// ---- __TESTs/MessagesTests/Complex/FB_ComplexDataTests.TcPOU
FUNCTION_BLOCK INTERNAL FINAL FB_ComplexDataTests EXTENDS FB_TestSuite
VAR
	fbVerify			: FB_TcUnitAdapter;
	fbVerifyBuffer 		: FB_TcUnitAdapter;
	fbWriterSUT			: FB_ComplexData;
	fbParserSUT			: FB_ComplexData;
	stActual			: ST_ComplexData;
	aBuffer				: ARRAY[0..255] OF BYTE;
	eTestState			: (DATA, BUFFER);
END_VAR
VAR CONSTANT
	cExpected			: ST_ComplexData := (label:= 'test-label 🐞!', value_dint:= -1, value_int:= -2, value_word:= 2,
											raw_bytes:= [44,33,22], raw_bytes_count:= 3,
											readings:= [(value:= 12345.67892, precision:= 2.3, timestamp:= 12345678), (value:= 999.888, precision:= 0.111, timestamp:= 777666555)], readings_count:= 2,
											data_type:= E_DataType.DATA_TYPE_TEMPERATURE);
END_VAR

VerifyData();
VerifyBuffer();

METHOD PRIVATE VerifyBuffer
VAR
	hr : HRESULT;
END_VAR
TEST(__POUNAME());

IF eTestState <> BUFFER THEN
	RETURN;
END_IF

hr := fbVerifyBuffer.Verify(anyArg:= aBuffer);

IF NOT PENDING(hr) THEN	
	TEST_FINISHED_NAMED(__POUNAME());
END_IF
END_METHOD

METHOD PRIVATE VerifyData
VAR_INST
	hr, hrWriter, hrParser : HRESULT;
	bOnce : BOOL := TRUE;
END_VAR
TEST(__POUNAME());
IF eTestState <> DATA THEN
	RETURN;
END_IF

// ARRANGE
fbWriterSUT.ComplexData := cExpected;

// ACT
IF bOnce THEN
	bOnce := FALSE;
	hrWriter := fbWriterSUT.Writer.WriteTo(aBuffer);
	hrParser := fbParserSUT.Parser.ParseFrom(aBuffer);
	stActual := fbParserSUT.ComplexData;
END_IF;

// ASSERT
hr := fbVerify.Verify(anyArg:= stActual);

IF NOT PENDING(hr) THEN
	AssertEquals_DINT(Expected:= 0, Actual:= hrWriter, Message:= 'Writer failed');
	AssertEquals_DINT(Expected:= 0, Actual:= hrParser, Message:= 'Parser failed');
	TEST_FINISHED_NAMED(__POUNAME());
	eTestState := BUFFER;
END_IF
END_METHOD

END_FUNCTION_BLOCK

// ---- __TESTs/MessagesTests/Complex/_gen/FB_ComplexData.TcPOU
(*******************************************************************************
                          protoc-gen-twincat V0.0.0.0                           
                  https://github.com/TcHaxx/protoc-gen-twincat                  
*******************************************************************************)
{attribute 'no_explicit_call' := 'do not call this POU directly'}
{attribute 'no-analysis'}
// Another message demonstrating all field options
FUNCTION_BLOCK INTERNAL FINAL FB_ComplexData IMPLEMENTS I_Message
VAR
    _fbMessageParser : FB_MessageParser(ipMessage:= THIS^);
    _fbMessageWriter : FB_MessageWriter(ipMessage:= THIS^);
    _stComplexData : ST_ComplexData;
    // repeated uint32 array_data = 5;
    _fbFieldCodecId5 : FB_FieldCodecUint32(nTag:= 16#2A);
    _fbRepeatedId5 : FB_RepeatedField(anyArray:= F_ToAnyType(_stComplexData.array_data), anyFirstElem:= F_ToAnyType(_stComplexData.array_data[0]), ipFieldCodec:= _fbFieldCodecId5);
    // repeated SensorReading readings = 10;
    _fbFieldCodecId10 : FB_FieldCodecMessage(nTag:= 16#52, ipMessage:= _fbreadings);
    _fbRepeatedId10 : FB_RepeatedField(anyArray:= F_ToAnyType(_stComplexData.readings), anyFirstElem:= F_ToAnyType(_stComplexData.readings[0]), ipFieldCodec:= _fbFieldCodecId10);
    _fbreadings : FB_SensorReading;
    END_VAR

{attribute 'no-analysis'}
(* Calculates the size of this message in Protocol Buffer wire format, in bytes. *)
METHOD CalculateSize : UDINT
VAR
    nSize : UDINT;
    nRepeatedFieldSize : UDINT;
END_VAR
// string label = 1;
nSize := nSize + 1 + F_ComputeStringSize(anyString:= _stComplexData.label);
// int32 value_dint = 2;
nSize := nSize + 1 + F_ComputeInt32Size(anyDint:= _stComplexData.value_dint);
// int32 value_int = 3;
nSize := nSize + 1 + F_ComputeInt32Size(anyDint:= _stComplexData.value_int);
// uint32 value_word = 4;
nSize := nSize + 1 + F_ComputeUint32Size(anyUdint:= _stComplexData.value_word);
// repeated uint32 array_data = 5;
_fbRepeatedId5.nCount := _stComplexData.array_data_count;
_fbRepeatedId5.CalculateSize(nSize => nRepeatedFieldSize);
nSize := nSize + nRepeatedFieldSize;
// Status state = 6;
nSize := nSize + 1 + F_ComputeEnumSize(anyEnum:= _stComplexData.state);
// bytes raw_bytes = 7;
nSize := nSize + 1 + F_ComputeBytesSize(aBytes:= _stComplexData.raw_bytes, nCount:= _stComplexData.raw_bytes_count);
// double measurement = 8;
nSize := nSize + 1 + F_ComputeDoubleSize(fValue:= _stComplexData.measurement);
// float calibration_factor = 9;
nSize := nSize + 1 + F_ComputeFloatSize(fValue:= _stComplexData.calibration_factor);
// repeated SensorReading readings = 10;
_fbRepeatedId10.nCount := _stComplexData.readings_count;
_fbRepeatedId10.CalculateSize(nSize => nRepeatedFieldSize);
nSize := nSize + nRepeatedFieldSize;
// DataType data_type = 11;
nSize := nSize + 1 + F_ComputeEnumSize(anyEnum:= _stComplexData.data_type);
CalculateSize := nSize;
END_METHOD

PROPERTY PUBLIC ComplexData : ST_ComplexData
GET
ComplexData := _stComplexData;
END_GET
SET
_stComplexData := ComplexData;
// repeated SensorReading readings = 10;
_stComplexData.readings := ComplexData.readings;
END_SET
END_PROPERTY

(* Merges the data from the specified coded input stream with the current message.*)
{attribute 'no-analysis'}
METHOD MergeFrom : HRESULT
VAR_IN_OUT
    fbParseCtx : FB_ParseContext;
END_VAR
VAR
    nTag : UDINT;
END_VAR
_fbRepeatedId10.Initialize();
_fbRepeatedId5.Initialize();
REPEAT
MergeFrom := fbParseCtx.ReadTag(nTag=> nTag);
IF SUCCEEDED(MergeFrom) AND nTag = 0 THEN
    EXIT;
END_IF;

IF FAILED(MergeFrom) THEN
    RETURN;
END_IF

CASE nTag OF
    16#0A:    // string label = 1;
        MergeFrom := fbParseCtx.ReadString(anyStringOut:= _stComplexData.label); 
    16#10:    // int32 value_dint = 2;
        MergeFrom := fbParseCtx.ReadInt32(anyDint:= _stComplexData.value_dint); 
    16#18:    // int32 value_int = 3;
        MergeFrom := fbParseCtx.ReadInt32(anyDint:= _stComplexData.value_int); 
    16#20:    // uint32 value_word = 4;
        MergeFrom := fbParseCtx.ReadUint32(anyUdint:= _stComplexData.value_word); 
    16#2A:    // repeated uint32 array_data = 5;
        MergeFrom := _fbRepeatedId5.AddEntriesFrom(fbParseCtx:= fbParseCtx, ipFieldCodec:= _fbFieldCodecId5,nCount=> _stComplexData.array_data_count);
    16#30:    // Status state = 6;
        MergeFrom := fbParseCtx.ReadEnum(anyEnum:= _stComplexData.state); 
    16#3A:    // bytes raw_bytes = 7;
        MergeFrom := fbParseCtx.ReadBytes(aBytes:= _stComplexData.raw_bytes, nCount=> _stComplexData.raw_bytes_count); 
    16#41:    // double measurement = 8;
        MergeFrom := fbParseCtx.ReadDouble(fValue=> _stComplexData.measurement); 
    16#4D:    // float calibration_factor = 9;
        MergeFrom := fbParseCtx.ReadFloat(fValue=> _stComplexData.calibration_factor); 
    16#52:    // repeated SensorReading readings = 10;
        MergeFrom := _fbRepeatedId10.AddEntriesFrom(fbParseCtx:= fbParseCtx, ipFieldCodec:= _fbFieldCodecId10,nCount=> _stComplexData.readings_count);
    16#58:    // DataType data_type = 11;
        MergeFrom := fbParseCtx.ReadEnum(anyEnum:= _stComplexData.data_type); 
ELSE
    MergeFrom := fbParseCtx.SkipLastField();
END_CASE

UNTIL (FAILED(MergeFrom) OR nTag = 0)
END_REPEAT
END_METHOD

PROPERTY PUBLIC MessageValue : T_Any
GET
MessageValue := F_ToAnyType(anyArg:= _stComplexData);
END_GET
END_PROPERTY

PROPERTY PUBLIC Parser : REFERENCE TO FB_MessageParser
GET
Parser REF= THIS^._fbMessageParser;
END_GET
END_PROPERTY

(* Writer for this message.*)
PROPERTY PUBLIC Writer : REFERENCE TO FB_MessageWriter
GET
Writer REF= THIS^._fbMessageWriter;
END_GET
END_PROPERTY

(* Writes the data to the given coded output stream.*)
{attribute 'no-analysis'}
METHOD WriteTo : HRESULT
VAR_IN_OUT
	(* Coded output stream to write the data to. *)
	fbWriteCtx	: FB_WriteContext;
END_VAR
// string label = 1;
WriteTo := fbWriteCtx.WriteTag(1, E_WireType.LengthDelimited);
IF FAILED(WriteTo) THEN
    RETURN;
END_IF
WriteTo := fbWriteCtx.WriteString(sStringToWrite:= _stComplexData.label);
IF FAILED(WriteTo) THEN
    RETURN;
END_IF
// int32 value_dint = 2;
WriteTo := fbWriteCtx.WriteTag(2, E_WireType.Varint);
IF FAILED(WriteTo) THEN
    RETURN;
END_IF
WriteTo := fbWriteCtx.WriteInt32(anyDint:= _stComplexData.value_dint);
IF FAILED(WriteTo) THEN
    RETURN;
END_IF
// int32 value_int = 3;
WriteTo := fbWriteCtx.WriteTag(3, E_WireType.Varint);
IF FAILED(WriteTo) THEN
    RETURN;
END_IF
WriteTo := fbWriteCtx.WriteInt32(anyDint:= _stComplexData.value_int);
IF FAILED(WriteTo) THEN
    RETURN;
END_IF
// uint32 value_word = 4;
WriteTo := fbWriteCtx.WriteTag(4, E_WireType.Varint);
IF FAILED(WriteTo) THEN
    RETURN;
END_IF
WriteTo := fbWriteCtx.WriteUint32(anyUdint:= _stComplexData.value_word);
IF FAILED(WriteTo) THEN
    RETURN;
END_IF
// repeated uint32 array_data = 5;
WriteTo := _fbRepeatedId5.WriteToWithCount(fbWriteCtx:= fbWriteCtx, ipFieldCodec:= _fbFieldCodecId5, nCount:= _stComplexData.array_data_count);
IF FAILED(WriteTo) THEN
    RETURN;
END_IF
// Status state = 6;
WriteTo := fbWriteCtx.WriteTag(6, E_WireType.Varint);
IF FAILED(WriteTo) THEN
    RETURN;
END_IF
WriteTo := fbWriteCtx.WriteEnum(anyEnum:= _stComplexData.state);
IF FAILED(WriteTo) THEN
    RETURN;
END_IF
// bytes raw_bytes = 7;
WriteTo := fbWriteCtx.WriteTag(7, E_WireType.LengthDelimited);
IF FAILED(WriteTo) THEN
    RETURN;
END_IF
WriteTo := fbWriteCtx.WriteBytes(aBytes:= _stComplexData.raw_bytes, nCount:= _stComplexData.raw_bytes_count);
IF FAILED(WriteTo) THEN
    RETURN;
END_IF
// double measurement = 8;
WriteTo := fbWriteCtx.WriteTag(8, E_WireType.Fixed64);
IF FAILED(WriteTo) THEN
    RETURN;
END_IF
WriteTo := fbWriteCtx.WriteDouble(fValue:= _stComplexData.measurement);
IF FAILED(WriteTo) THEN
    RETURN;
END_IF
// float calibration_factor = 9;
WriteTo := fbWriteCtx.WriteTag(9, E_WireType.Fixed32);
IF FAILED(WriteTo) THEN
    RETURN;
END_IF
WriteTo := fbWriteCtx.WriteFloat(fValue:= _stComplexData.calibration_factor);
IF FAILED(WriteTo) THEN
    RETURN;
END_IF
// repeated SensorReading readings = 10;
WriteTo := _fbRepeatedId10.WriteToWithCount(fbWriteCtx:= fbWriteCtx, ipFieldCodec:= _fbFieldCodecId10, nCount:= _stComplexData.readings_count);
IF FAILED(WriteTo) THEN
    RETURN;
END_IF
// DataType data_type = 11;
WriteTo := fbWriteCtx.WriteTag(11, E_WireType.Varint);
IF FAILED(WriteTo) THEN
    RETURN;
END_IF
WriteTo := fbWriteCtx.WriteEnum(anyEnum:= _stComplexData.data_type);
IF FAILED(WriteTo) THEN
    RETURN;
END_IF
END_METHOD

END_FUNCTION_BLOCK

// ---- __TESTs/MessagesTests/Complex/_gen/FB_SensorReading.TcPOU
(*******************************************************************************
                          protoc-gen-twincat V0.0.0.0                           
                  https://github.com/TcHaxx/protoc-gen-twincat                  
*******************************************************************************)
{attribute 'no_explicit_call' := 'do not call this POU directly'}
{attribute 'no-analysis'}
FUNCTION_BLOCK INTERNAL FINAL FB_SensorReading IMPLEMENTS I_Message
VAR
    _fbMessageParser : FB_MessageParser(ipMessage:= THIS^);
    _fbMessageWriter : FB_MessageWriter(ipMessage:= THIS^);
    _stSensorReading : ST_SensorReading;
    END_VAR

{attribute 'no-analysis'}
(* Calculates the size of this message in Protocol Buffer wire format, in bytes. *)
METHOD CalculateSize : UDINT
VAR
    nSize : UDINT;
    nRepeatedFieldSize : UDINT;
END_VAR
// double value = 1;
nSize := nSize + 1 + F_ComputeDoubleSize(fValue:= _stSensorReading.value);
// float precision = 2;
nSize := nSize + 1 + F_ComputeFloatSize(fValue:= _stSensorReading.precision);
// int64 timestamp = 3;
nSize := nSize + 1 + F_ComputeInt64Size(anyLint:= _stSensorReading.timestamp);
CalculateSize := nSize;
END_METHOD

(* Merges the data from the specified coded input stream with the current message.*)
{attribute 'no-analysis'}
METHOD MergeFrom : HRESULT
VAR_IN_OUT
    fbParseCtx : FB_ParseContext;
END_VAR
VAR
    nTag : UDINT;
END_VAR
REPEAT
MergeFrom := fbParseCtx.ReadTag(nTag=> nTag);
IF SUCCEEDED(MergeFrom) AND nTag = 0 THEN
    EXIT;
END_IF;

IF FAILED(MergeFrom) THEN
    RETURN;
END_IF

CASE nTag OF
    16#09:    // double value = 1;
        MergeFrom := fbParseCtx.ReadDouble(fValue=> _stSensorReading.value); 
    16#15:    // float precision = 2;
        MergeFrom := fbParseCtx.ReadFloat(fValue=> _stSensorReading.precision); 
    16#18:    // int64 timestamp = 3;
        MergeFrom := fbParseCtx.ReadInt64(anyLint:= _stSensorReading.timestamp); 
ELSE
    MergeFrom := fbParseCtx.SkipLastField();
END_CASE

UNTIL (FAILED(MergeFrom) OR nTag = 0)
END_REPEAT
END_METHOD

PROPERTY PUBLIC MessageValue : T_Any
GET
MessageValue := F_ToAnyType(anyArg:= _stSensorReading);
END_GET
END_PROPERTY

PROPERTY PUBLIC Parser : REFERENCE TO FB_MessageParser
GET
Parser REF= THIS^._fbMessageParser;
END_GET
END_PROPERTY

PROPERTY PUBLIC SensorReading : ST_SensorReading
GET
SensorReading := _stSensorReading;
END_GET
SET
_stSensorReading := SensorReading;
END_SET
END_PROPERTY

(* Writer for this message.*)
PROPERTY PUBLIC Writer : REFERENCE TO FB_MessageWriter
GET
Writer REF= THIS^._fbMessageWriter;
END_GET
END_PROPERTY

(* Writes the data to the given coded output stream.*)
{attribute 'no-analysis'}
METHOD WriteTo : HRESULT
VAR_IN_OUT
	(* Coded output stream to write the data to. *)
	fbWriteCtx	: FB_WriteContext;
END_VAR
// double value = 1;
WriteTo := fbWriteCtx.WriteTag(1, E_WireType.Fixed64);
IF FAILED(WriteTo) THEN
    RETURN;
END_IF
WriteTo := fbWriteCtx.WriteDouble(fValue:= _stSensorReading.value);
IF FAILED(WriteTo) THEN
    RETURN;
END_IF
// float precision = 2;
WriteTo := fbWriteCtx.WriteTag(2, E_WireType.Fixed32);
IF FAILED(WriteTo) THEN
    RETURN;
END_IF
WriteTo := fbWriteCtx.WriteFloat(fValue:= _stSensorReading.precision);
IF FAILED(WriteTo) THEN
    RETURN;
END_IF
// int64 timestamp = 3;
WriteTo := fbWriteCtx.WriteTag(3, E_WireType.Varint);
IF FAILED(WriteTo) THEN
    RETURN;
END_IF
WriteTo := fbWriteCtx.WriteInt64(anyLint:= _stSensorReading.timestamp);
IF FAILED(WriteTo) THEN
    RETURN;
END_IF
END_METHOD

END_FUNCTION_BLOCK

// ---- POUs/ComputeSize/F_ComputeEnumSize.TcPOU
FUNCTION F_ComputeEnumSize : UDINT
VAR_INPUT
    anyEnum  : ANY;
END_VAR
VAR
	nTmp : DINT;
END_VAR

IF anyEnum.pValue = NULL OR anyEnum.TypeClass <> __SYSTEM.TYPE_CLASS.TYPE_ENUM THEN
	RETURN;
END_IF

MEMCPY(destAddr:= ADR(nTmp), srcAddr:= anyEnum.pValue, MIN(TO_UDINT(anyEnum.diSize), SIZEOF(nTmp)));
F_ComputeEnumSize := F_ComputeInt32Size(nTmp);

END_FUNCTION

// ---- __TESTs/MessagesTests/Complex/FB_RepeatedComplexDataTests.TcPOU
FUNCTION_BLOCK INTERNAL FINAL FB_RepeatedComplexDataTests EXTENDS FB_TestSuite
VAR
	fbVerify			: FB_TcUnitAdapter;
	fbVerifyBuffer 		: FB_TcUnitAdapter;
	fbWriterSUT			: FB_RepeatedComplexData;
	fbParserSUT			: FB_RepeatedComplexData;
	stActual			: ST_RepeatedComplexData;
	aBuffer				: ARRAY[0..4095] OF BYTE;
	eTestState			: (DATA, BUFFER);
	lenMsg, nBufferPos : UDINT;
END_VAR
VAR CONSTANT
	cExpected			: ST_RepeatedComplexData := (
						    complex_data_list_count := 1,
							complex_data_list := [(label:= 'test-label 🐞!', value_dint:= -1, value_int:= -2, value_word:= 2,
											raw_bytes:= [44,33,22], raw_bytes_count:= 3,
											array_data:= [123, 42, 69],
											array_data_count := 3,
											readings:= [(value:= 12345.67892, precision:= 2.3, timestamp:= 12345678), (value:= 999.888, precision:= 0.111, timestamp:= 777666555)], readings_count:= 2,
											data_type:= E_DataType.DATA_TYPE_TEMPERATURE)]);
END_VAR

VerifyData();
VerifyBuffer();

fbWriterSUT.RepeatedComplexData := cExpected;
lenMsg := fbWriterSUT.CalculateSize();
fbWriterSUT.Writer.WriteTo(aBuffer);

nBufferPos := fbWriterSUT.Writer.fbWriteCtx.refCtx.stState.nBufferPos;

METHOD PRIVATE VerifyBuffer
VAR
	hr : HRESULT;
END_VAR
TEST(__POUNAME());

IF eTestState <> BUFFER THEN
	RETURN;
END_IF

hr := fbVerifyBuffer.Verify(anyArg:= aBuffer);

IF NOT PENDING(hr) THEN	
	TEST_FINISHED_NAMED(__POUNAME());
END_IF
END_METHOD

METHOD PRIVATE VerifyData
VAR_INST
	hr, hrWriter, hrParser : HRESULT := S_PENDING;
	bOnce : BOOL := TRUE;
END_VAR
TEST(__POUNAME());
IF eTestState <> DATA THEN
	RETURN;
END_IF

// ARRANGE
fbWriterSUT.RepeatedComplexData := cExpected;

// ACT
IF bOnce THEN
	bOnce := FALSE;
	hrWriter := fbWriterSUT.Writer.WriteTo(aBuffer);
	hrParser := fbParserSUT.Parser.ParseFrom(aBuffer);
	stActual := fbParserSUT.RepeatedComplexData;
END_IF;

// ASSERT
hr := fbVerify.Verify(anyArg:= stActual);

IF NOT PENDING(hr) THEN
	AssertEquals_DINT(Expected:= 0, Actual:= hrWriter, Message:= 'Writer failed');
	AssertEquals_DINT(Expected:= 0, Actual:= hrParser, Message:= 'Parser failed');
	TEST_FINISHED_NAMED(__POUNAME());
	eTestState := BUFFER;
END_IF
END_METHOD

END_FUNCTION_BLOCK

// ---- __TESTs/MessagesTests/Complex/_gen/FB_RepeatedComplexData.TcPOU
(*******************************************************************************
                          protoc-gen-twincat V0.0.0.0                           
                  https://github.com/TcHaxx/protoc-gen-twincat                  
*******************************************************************************)
{attribute 'no_explicit_call' := 'do not call this POU directly'}
{attribute 'no-analysis'}
FUNCTION_BLOCK INTERNAL FINAL FB_RepeatedComplexData IMPLEMENTS I_Message
VAR
    _fbMessageParser : FB_MessageParser(ipMessage:= THIS^);
    _fbMessageWriter : FB_MessageWriter(ipMessage:= THIS^);
    _stRepeatedComplexData : ST_RepeatedComplexData;
    // repeated ComplexData complex_data_list = 1;
    _fbFieldCodecId1 : FB_FieldCodecMessage(nTag:= 16#0A, ipMessage:= _fbcomplex_data_list);
    _fbRepeatedId1 : FB_RepeatedField(anyArray:= F_ToAnyType(_stRepeatedComplexData.complex_data_list), anyFirstElem:= F_ToAnyType(_stRepeatedComplexData.complex_data_list[0]), ipFieldCodec:= _fbFieldCodecId1);
    _fbcomplex_data_list : FB_ComplexData;
    END_VAR

{attribute 'no-analysis'}
(* Calculates the size of this message in Protocol Buffer wire format, in bytes. *)
METHOD CalculateSize : UDINT
VAR
    nSize : UDINT;
    nRepeatedFieldSize : UDINT;
END_VAR
// repeated ComplexData complex_data_list = 1;
_fbRepeatedId1.nCount := _stRepeatedComplexData.complex_data_list_count;
_fbRepeatedId1.CalculateSize(nSize => nRepeatedFieldSize);
nSize := nSize + nRepeatedFieldSize;
CalculateSize := nSize;
END_METHOD

(* Merges the data from the specified coded input stream with the current message.*)
{attribute 'no-analysis'}
METHOD MergeFrom : HRESULT
VAR_IN_OUT
    fbParseCtx : FB_ParseContext;
END_VAR
VAR
    nTag : UDINT;
END_VAR
_fbRepeatedId1.Initialize();
REPEAT
MergeFrom := fbParseCtx.ReadTag(nTag=> nTag);
IF SUCCEEDED(MergeFrom) AND nTag = 0 THEN
    EXIT;
END_IF;

IF FAILED(MergeFrom) THEN
    RETURN;
END_IF

CASE nTag OF
    16#0A:    // repeated ComplexData complex_data_list = 1;
        MergeFrom := _fbRepeatedId1.AddEntriesFrom(fbParseCtx:= fbParseCtx, ipFieldCodec:= _fbFieldCodecId1,nCount=> _stRepeatedComplexData.complex_data_list_count);
ELSE
    MergeFrom := fbParseCtx.SkipLastField();
END_CASE

UNTIL (FAILED(MergeFrom) OR nTag = 0)
END_REPEAT
END_METHOD

PROPERTY PUBLIC MessageValue : T_Any
GET
MessageValue := F_ToAnyType(anyArg:= _stRepeatedComplexData);
END_GET
END_PROPERTY

PROPERTY PUBLIC Parser : REFERENCE TO FB_MessageParser
GET
Parser REF= THIS^._fbMessageParser;
END_GET
END_PROPERTY

PROPERTY PUBLIC RepeatedComplexData : ST_RepeatedComplexData
GET
RepeatedComplexData := _stRepeatedComplexData;
END_GET
SET
_stRepeatedComplexData := RepeatedComplexData;
// repeated ComplexData complex_data_list = 1;
_stRepeatedComplexData.complex_data_list := RepeatedComplexData.complex_data_list;
END_SET
END_PROPERTY

(* Writer for this message.*)
PROPERTY PUBLIC Writer : REFERENCE TO FB_MessageWriter
GET
Writer REF= THIS^._fbMessageWriter;
END_GET
END_PROPERTY

(* Writes the data to the given coded output stream.*)
{attribute 'no-analysis'}
METHOD WriteTo : HRESULT
VAR_IN_OUT
	(* Coded output stream to write the data to. *)
	fbWriteCtx	: FB_WriteContext;
END_VAR
// repeated ComplexData complex_data_list = 1;
WriteTo := _fbRepeatedId1.WriteToWithCount(fbWriteCtx:= fbWriteCtx, ipFieldCodec:= _fbFieldCodecId1, nCount:= _stRepeatedComplexData.complex_data_list_count);
IF FAILED(WriteTo) THEN
    RETURN;
END_IF
END_METHOD

END_FUNCTION_BLOCK

// ---- __TESTs/MessagesTests/Complex/FB_MotorTests.TcPOU
FUNCTION_BLOCK INTERNAL FINAL FB_MotorTests EXTENDS FB_TestSuite
VAR
	fbVerify			: FB_TcUnitAdapter;
	fbVerifyBuffer 		: FB_TcUnitAdapter;
	fbWriterSUT			: FB_Motor;
	fbParserSUT			: FB_Motor;
	stActual			: ST_Motor;
	aBuffer				: ARRAY[0..255] OF BYTE;
	eTestState			: (DATA, BUFFER);
END_VAR
VAR CONSTANT
	cExpected			: ST_Motor := (name:= 'test-name 🐞!', status:= E_Status.STATUS_RUNNING, speed:= 16#1234,
									   sensor_readings:= [1,2,3,4,5,6,7,8], sensor_readings_count:= 8,
									   config:= [9,8,7], config_count:= 3,
									   motor_config:= (max_speed:= 123.567, acceleration:= 567.123, timeout_ms:= 42));
END_VAR

VerifyData();
VerifyBuffer();

METHOD PRIVATE VerifyBuffer
VAR
	hr : HRESULT;
END_VAR
TEST(__POUNAME());

IF eTestState <> BUFFER THEN
	RETURN;
END_IF

hr := fbVerifyBuffer.Verify(anyArg:= aBuffer);

IF NOT PENDING(hr) THEN	
	TEST_FINISHED_NAMED(__POUNAME());
END_IF
END_METHOD

METHOD PRIVATE VerifyData
VAR
	hr, hrWriter, hrParser : HRESULT;
END_VAR
TEST(__POUNAME());
IF eTestState <> DATA THEN
	RETURN;
END_IF

// ARRANGE
fbWriterSUT.Motor := cExpected;

// ACT
hrWriter := fbWriterSUT.Writer.WriteTo(aBuffer);
hrParser := fbParserSUT.Parser.ParseFrom(aBuffer);
stActual := fbParserSUT.Motor;

// ASSERT
hr := fbVerify.Verify(anyArg:= stActual);

IF NOT PENDING(hr) THEN
	AssertEquals_DINT(Expected:= 0, Actual:= hrWriter, Message:= '');
	AssertEquals_DINT(Expected:= 0, Actual:= hrParser, Message:= '');
	TEST_FINISHED_NAMED(__POUNAME());
	eTestState := BUFFER;
END_IF
END_METHOD

END_FUNCTION_BLOCK

// ---- __TESTs/MessagesTests/Complex/_gen/FB_Motor.TcPOU
(*******************************************************************************
                          protoc-gen-twincat V0.0.0.0                           
                  https://github.com/TcHaxx/protoc-gen-twincat                  
*******************************************************************************)
{attribute 'no_explicit_call' := 'do not call this POU directly'}
{attribute 'no-analysis'}
// Message with fb_prefix option (function block)
FUNCTION_BLOCK INTERNAL FINAL FB_Motor IMPLEMENTS I_Message
VAR
    _fbMessageParser : FB_MessageParser(ipMessage:= THIS^);
    _fbMessageWriter : FB_MessageWriter(ipMessage:= THIS^);
    _stMotor : ST_Motor;
    // repeated int32 sensor_readings = 4;
    _fbFieldCodecId4 : FB_FieldCodecInt32(nTag:= 16#22);
    _fbRepeatedId4 : FB_RepeatedField(anyArray:= F_ToAnyType(_stMotor.sensor_readings), anyFirstElem:= F_ToAnyType(_stMotor.sensor_readings[0]), ipFieldCodec:= _fbFieldCodecId4);
    _fbmotor_config : FB_MotorConfig;
    END_VAR

{attribute 'no-analysis'}
(* Calculates the size of this message in Protocol Buffer wire format, in bytes. *)
METHOD CalculateSize : UDINT
VAR
    nSize : UDINT;
    nRepeatedFieldSize : UDINT;
END_VAR
// string name = 1;
nSize := nSize + 1 + F_ComputeStringSize(anyString:= _stMotor.name);
// Status status = 2;
nSize := nSize + 1 + F_ComputeEnumSize(anyEnum:= _stMotor.status);
// uint32 speed = 3;
nSize := nSize + 1 + F_ComputeUint32Size(anyUdint:= _stMotor.speed);
// repeated int32 sensor_readings = 4;
_fbRepeatedId4.nCount := _stMotor.sensor_readings_count;
_fbRepeatedId4.CalculateSize(nSize => nRepeatedFieldSize);
nSize := nSize + nRepeatedFieldSize;
// bytes config = 5;
nSize := nSize + 1 + F_ComputeBytesSize(aBytes:= _stMotor.config, nCount:= _stMotor.config_count);
// MotorConfig motor_config = 6;
nSize := nSize + 1 + F_ComputeMessageSize(iMessage:= _fbmotor_config);
CalculateSize := nSize;
END_METHOD

(* Merges the data from the specified coded input stream with the current message.*)
{attribute 'no-analysis'}
METHOD MergeFrom : HRESULT
VAR_IN_OUT
    fbParseCtx : FB_ParseContext;
END_VAR
VAR
    nTag : UDINT;
END_VAR
_fbRepeatedId4.Initialize();
REPEAT
MergeFrom := fbParseCtx.ReadTag(nTag=> nTag);
IF SUCCEEDED(MergeFrom) AND nTag = 0 THEN
    EXIT;
END_IF;

IF FAILED(MergeFrom) THEN
    RETURN;
END_IF

CASE nTag OF
    16#0A:    // string name = 1;
        MergeFrom := fbParseCtx.ReadString(anyStringOut:= _stMotor.name); 
    16#10:    // Status status = 2;
        MergeFrom := fbParseCtx.ReadEnum(anyEnum:= _stMotor.status); 
    16#18:    // uint32 speed = 3;
        MergeFrom := fbParseCtx.ReadUint32(anyUdint:= _stMotor.speed); 
    16#22:    // repeated int32 sensor_readings = 4;
        MergeFrom := _fbRepeatedId4.AddEntriesFrom(fbParseCtx:= fbParseCtx, ipFieldCodec:= _fbFieldCodecId4,nCount=> _stMotor.sensor_readings_count);
    16#2A:    // bytes config = 5;
        MergeFrom := fbParseCtx.ReadBytes(aBytes:= _stMotor.config, nCount=> _stMotor.config_count); 
    16#32:    // MotorConfig motor_config = 6;
        MergeFrom := fbParseCtx.ReadMessage(ipMessage:= _fbmotor_config);
        THIS^._stMotor.motor_config := _fbmotor_config.MotorConfig;
ELSE
    MergeFrom := fbParseCtx.SkipLastField();
END_CASE

UNTIL (FAILED(MergeFrom) OR nTag = 0)
END_REPEAT
END_METHOD

PROPERTY PUBLIC MessageValue : T_Any
GET
MessageValue := F_ToAnyType(anyArg:= _stMotor);
END_GET
END_PROPERTY

PROPERTY PUBLIC Motor : ST_Motor
GET
Motor := _stMotor;
END_GET
SET
_stMotor := Motor;
// MotorConfig motor_config = 6;
_stMotor.motor_config := Motor.motor_config;
END_SET
END_PROPERTY

PROPERTY PUBLIC Parser : REFERENCE TO FB_MessageParser
GET
Parser REF= THIS^._fbMessageParser;
END_GET
END_PROPERTY

(* Writer for this message.*)
PROPERTY PUBLIC Writer : REFERENCE TO FB_MessageWriter
GET
Writer REF= THIS^._fbMessageWriter;
END_GET
END_PROPERTY

(* Writes the data to the given coded output stream.*)
{attribute 'no-analysis'}
METHOD WriteTo : HRESULT
VAR_IN_OUT
	(* Coded output stream to write the data to. *)
	fbWriteCtx	: FB_WriteContext;
END_VAR
// string name = 1;
WriteTo := fbWriteCtx.WriteTag(1, E_WireType.LengthDelimited);
IF FAILED(WriteTo) THEN
    RETURN;
END_IF
WriteTo := fbWriteCtx.WriteString(sStringToWrite:= _stMotor.name);
IF FAILED(WriteTo) THEN
    RETURN;
END_IF
// Status status = 2;
WriteTo := fbWriteCtx.WriteTag(2, E_WireType.Varint);
IF FAILED(WriteTo) THEN
    RETURN;
END_IF
WriteTo := fbWriteCtx.WriteEnum(anyEnum:= _stMotor.status);
IF FAILED(WriteTo) THEN
    RETURN;
END_IF
// uint32 speed = 3;
WriteTo := fbWriteCtx.WriteTag(3, E_WireType.Varint);
IF FAILED(WriteTo) THEN
    RETURN;
END_IF
WriteTo := fbWriteCtx.WriteUint32(anyUdint:= _stMotor.speed);
IF FAILED(WriteTo) THEN
    RETURN;
END_IF
// repeated int32 sensor_readings = 4;
WriteTo := _fbRepeatedId4.WriteToWithCount(fbWriteCtx:= fbWriteCtx, ipFieldCodec:= _fbFieldCodecId4, nCount:= _stMotor.sensor_readings_count);
IF FAILED(WriteTo) THEN
    RETURN;
END_IF
// bytes config = 5;
WriteTo := fbWriteCtx.WriteTag(5, E_WireType.LengthDelimited);
IF FAILED(WriteTo) THEN
    RETURN;
END_IF
WriteTo := fbWriteCtx.WriteBytes(aBytes:= _stMotor.config, nCount:= _stMotor.config_count);
IF FAILED(WriteTo) THEN
    RETURN;
END_IF
// MotorConfig motor_config = 6;
WriteTo := fbWriteCtx.WriteTag(6, E_WireType.LengthDelimited);
IF FAILED(WriteTo) THEN
    RETURN;
END_IF
_fbmotor_config.MotorConfig := THIS^._stMotor.motor_config;
WriteTo := fbWriteCtx.WriteMessage(ipMessage:= THIS^._fbmotor_config);
IF FAILED(WriteTo) THEN
    RETURN;
END_IF
END_METHOD

END_FUNCTION_BLOCK

// ---- FieldCodec/FB_FieldCodecInt32.TcPOU
FUNCTION_BLOCK FB_FieldCodecInt32 EXTENDS FB_FieldCodec
VAR_INPUT
END_VAR
VAR_OUTPUT
END_VAR
VAR
    nValue : DINT;
END_VAR

METHOD CalculatePackedDataSize : HRESULT
VAR_INPUT CONSTANT
	anyFirstElem	: T_Any;
	nLength	        : UDINT;        // items to write
END_VAR
VAR_OUTPUT
    nPackedDataSize : UDINT;
END_VAR
VAR
    anyItem         : T_ANY;
    i               : UDINT;
    nValue          : DINT;
END_VAR
anyItem := anyFirstElem;

IF nLength < 1 THEN
    nPackedDataSize := 0;
    RETURN;
END_IF

FOR i := 0  TO nLength - 1 DO
    anyItem.pValue := anyFirstElem.pValue + (i * TO_UDINT(anyFirstElem.diSize)); 
    nValue := PDINT_TO_DINT(anyItem.pValue);
    nPackedDataSize := nPackedDataSize + F_ComputeInt32Size(nValue);
END_FOR
END_METHOD

METHOD IsPackedRepeatedField : BOOL
VAR_INPUT
	nTag	: UDINT;
END_VAR
IsPackedRepeatedField := F_IsPackedRepeatedField(nTag);
END_METHOD


METHOD ValueReader : HRESULT
VAR_IN_OUT      
    stCtx : ST_ParseContext;
END_VAR
VAR_OUTPUT
	anyOut	: T_Any;
END_VAR

ValueReader := F_ParseRawVarint32(stCtx, nValue);
anyOut := F_ToAnyType(anyArg:= nValue);
END_METHOD

METHOD ValueWriter : HRESULT
VAR_IN_OUT
    stCtx  : ST_WriteContext;
END_VAR
VAR_INPUT
    anyIn : T_ANY;
END_VAR
VAR
    nValue  : DINT;
END_VAR

nValue := PDINT_TO_DINT(anyIn.pValue);
ValueWriter := F_WriteInt32(stCtx, nValue);
END_METHOD

END_FUNCTION_BLOCK

// ---- __TESTs/MessagesTests/Complex/_gen/FB_MotorConfig.TcPOU
(*******************************************************************************
                          protoc-gen-twincat V0.0.0.0                           
                  https://github.com/TcHaxx/protoc-gen-twincat                  
*******************************************************************************)
{attribute 'no_explicit_call' := 'do not call this POU directly'}
{attribute 'no-analysis'}
FUNCTION_BLOCK INTERNAL FINAL FB_MotorConfig IMPLEMENTS I_Message
VAR
    _fbMessageParser : FB_MessageParser(ipMessage:= THIS^);
    _fbMessageWriter : FB_MessageWriter(ipMessage:= THIS^);
    _stMotorConfig : ST_MotorConfig;
    END_VAR

{attribute 'no-analysis'}
(* Calculates the size of this message in Protocol Buffer wire format, in bytes. *)
METHOD CalculateSize : UDINT
VAR
    nSize : UDINT;
    nRepeatedFieldSize : UDINT;
END_VAR
// float max_speed = 1;
nSize := nSize + 1 + F_ComputeFloatSize(fValue:= _stMotorConfig.max_speed);
// double acceleration = 2;
nSize := nSize + 1 + F_ComputeDoubleSize(fValue:= _stMotorConfig.acceleration);
// uint32 timeout_ms = 3;
nSize := nSize + 1 + F_ComputeUint32Size(anyUdint:= _stMotorConfig.timeout_ms);
CalculateSize := nSize;
END_METHOD

(* Merges the data from the specified coded input stream with the current message.*)
{attribute 'no-analysis'}
METHOD MergeFrom : HRESULT
VAR_IN_OUT
    fbParseCtx : FB_ParseContext;
END_VAR
VAR
    nTag : UDINT;
END_VAR
REPEAT
MergeFrom := fbParseCtx.ReadTag(nTag=> nTag);
IF SUCCEEDED(MergeFrom) AND nTag = 0 THEN
    EXIT;
END_IF;

IF FAILED(MergeFrom) THEN
    RETURN;
END_IF

CASE nTag OF
    16#0D:    // float max_speed = 1;
        MergeFrom := fbParseCtx.ReadFloat(fValue=> _stMotorConfig.max_speed); 
    16#11:    // double acceleration = 2;
        MergeFrom := fbParseCtx.ReadDouble(fValue=> _stMotorConfig.acceleration); 
    16#18:    // uint32 timeout_ms = 3;
        MergeFrom := fbParseCtx.ReadUint32(anyUdint:= _stMotorConfig.timeout_ms); 
ELSE
    MergeFrom := fbParseCtx.SkipLastField();
END_CASE

UNTIL (FAILED(MergeFrom) OR nTag = 0)
END_REPEAT
END_METHOD

PROPERTY PUBLIC MessageValue : T_Any
GET
MessageValue := F_ToAnyType(anyArg:= _stMotorConfig);
END_GET
END_PROPERTY

PROPERTY PUBLIC MotorConfig : ST_MotorConfig
GET
MotorConfig := _stMotorConfig;
END_GET
SET
_stMotorConfig := MotorConfig;
END_SET
END_PROPERTY

PROPERTY PUBLIC Parser : REFERENCE TO FB_MessageParser
GET
Parser REF= THIS^._fbMessageParser;
END_GET
END_PROPERTY

(* Writer for this message.*)
PROPERTY PUBLIC Writer : REFERENCE TO FB_MessageWriter
GET
Writer REF= THIS^._fbMessageWriter;
END_GET
END_PROPERTY

(* Writes the data to the given coded output stream.*)
{attribute 'no-analysis'}
METHOD WriteTo : HRESULT
VAR_IN_OUT
	(* Coded output stream to write the data to. *)
	fbWriteCtx	: FB_WriteContext;
END_VAR
// float max_speed = 1;
WriteTo := fbWriteCtx.WriteTag(1, E_WireType.Fixed32);
IF FAILED(WriteTo) THEN
    RETURN;
END_IF
WriteTo := fbWriteCtx.WriteFloat(fValue:= _stMotorConfig.max_speed);
IF FAILED(WriteTo) THEN
    RETURN;
END_IF
// double acceleration = 2;
WriteTo := fbWriteCtx.WriteTag(2, E_WireType.Fixed64);
IF FAILED(WriteTo) THEN
    RETURN;
END_IF
WriteTo := fbWriteCtx.WriteDouble(fValue:= _stMotorConfig.acceleration);
IF FAILED(WriteTo) THEN
    RETURN;
END_IF
// uint32 timeout_ms = 3;
WriteTo := fbWriteCtx.WriteTag(3, E_WireType.Varint);
IF FAILED(WriteTo) THEN
    RETURN;
END_IF
WriteTo := fbWriteCtx.WriteUint32(anyUdint:= _stMotorConfig.timeout_ms);
IF FAILED(WriteTo) THEN
    RETURN;
END_IF
END_METHOD

END_FUNCTION_BLOCK

// ---- __TESTs/MessagesTests/Complex/FB_DeviceTests.TcPOU
FUNCTION_BLOCK INTERNAL FINAL FB_DeviceTests EXTENDS FB_TestSuite
VAR
	fbVerify			: FB_TcUnitAdapter;
	fbVerifyBuffer 		: FB_TcUnitAdapter;
	fbWriterSUT			: FB_Device;
	fbParserSUT			: FB_Device;
	stActual			: ST_Device;
	aBuffer				: ARRAY[0..255] OF BYTE;
	eTestState			: (DATA, BUFFER);
END_VAR
VAR CONSTANT
	cExpected			: ST_Device := (name:= 'test-name ⚠️!', id:= 16#1234,
									   error_codes:= [1,2,3,4,5,6,7,8,9,10], error_codes_count:= 10,
									   temperature:= -3,
									   data:= [62(16#CC), 13,37], data_count:= 64);
END_VAR

VerifyData();
VerifyBuffer();

METHOD PRIVATE VerifyBuffer
VAR
	hr : HRESULT;
END_VAR
TEST(__POUNAME());

IF eTestState <> BUFFER THEN
	RETURN;
END_IF

hr := fbVerifyBuffer.Verify(anyArg:= aBuffer);

IF NOT PENDING(hr) THEN	
	TEST_FINISHED_NAMED(__POUNAME());
END_IF
END_METHOD

METHOD PRIVATE VerifyData
VAR
	hr, hrWriter, hrParser : HRESULT;
END_VAR
TEST(__POUNAME());
IF eTestState <> DATA THEN
	RETURN;
END_IF

// ARRANGE
fbWriterSUT.Device := cExpected;

// ACT
hrWriter := fbWriterSUT.Writer.WriteTo(aBuffer);
hrParser := fbParserSUT.Parser.ParseFrom(aBuffer);
stActual := fbParserSUT.Device;

// ASSERT
hr := fbVerify.Verify(anyArg:= stActual);

IF NOT PENDING(hr) THEN
	AssertEquals_DINT(Expected:= 0, Actual:= hrWriter, Message:= '');
	AssertEquals_DINT(Expected:= 0, Actual:= hrParser, Message:= '');
	TEST_FINISHED_NAMED(__POUNAME());
	eTestState := BUFFER;
END_IF
END_METHOD

END_FUNCTION_BLOCK

// ---- __TESTs/MessagesTests/Complex/_gen/FB_Device.TcPOU
(*******************************************************************************
                          protoc-gen-twincat V0.0.0.0                           
                  https://github.com/TcHaxx/protoc-gen-twincat                  
*******************************************************************************)
{attribute 'no_explicit_call' := 'do not call this POU directly'}
{attribute 'no-analysis'}
// Message with st_prefix and attribute_pack_mode options
FUNCTION_BLOCK INTERNAL FINAL FB_Device IMPLEMENTS I_Message
VAR
    _fbMessageParser : FB_MessageParser(ipMessage:= THIS^);
    _fbMessageWriter : FB_MessageWriter(ipMessage:= THIS^);
    _stDevice : ST_Device;
    // repeated uint32 error_codes = 3;
    _fbFieldCodecId3 : FB_FieldCodecUint32(nTag:= 16#1A);
    _fbRepeatedId3 : FB_RepeatedField(anyArray:= F_ToAnyType(_stDevice.error_codes), anyFirstElem:= F_ToAnyType(_stDevice.error_codes[0]), ipFieldCodec:= _fbFieldCodecId3);
    END_VAR

{attribute 'no-analysis'}
(* Calculates the size of this message in Protocol Buffer wire format, in bytes. *)
METHOD CalculateSize : UDINT
VAR
    nSize : UDINT;
    nRepeatedFieldSize : UDINT;
END_VAR
// string name = 1;
nSize := nSize + 1 + F_ComputeStringSize(anyString:= _stDevice.name);
// uint32 id = 2;
nSize := nSize + 1 + F_ComputeUint32Size(anyUdint:= _stDevice.id);
// repeated uint32 error_codes = 3;
_fbRepeatedId3.nCount := _stDevice.error_codes_count;
_fbRepeatedId3.CalculateSize(nSize => nRepeatedFieldSize);
nSize := nSize + nRepeatedFieldSize;
// int32 temperature = 4;
nSize := nSize + 1 + F_ComputeInt32Size(anyDint:= _stDevice.temperature);
// bytes data = 5;
nSize := nSize + 1 + F_ComputeBytesSize(aBytes:= _stDevice.data, nCount:= _stDevice.data_count);
CalculateSize := nSize;
END_METHOD

PROPERTY PUBLIC Device : ST_Device
GET
Device := _stDevice;
END_GET
SET
_stDevice := Device;
END_SET
END_PROPERTY

(* Merges the data from the specified coded input stream with the current message.*)
{attribute 'no-analysis'}
METHOD MergeFrom : HRESULT
VAR_IN_OUT
    fbParseCtx : FB_ParseContext;
END_VAR
VAR
    nTag : UDINT;
END_VAR
_fbRepeatedId3.Initialize();
REPEAT
MergeFrom := fbParseCtx.ReadTag(nTag=> nTag);
IF SUCCEEDED(MergeFrom) AND nTag = 0 THEN
    EXIT;
END_IF;

IF FAILED(MergeFrom) THEN
    RETURN;
END_IF

CASE nTag OF
    16#0A:    // string name = 1;
        MergeFrom := fbParseCtx.ReadString(anyStringOut:= _stDevice.name); 
    16#10:    // uint32 id = 2;
        MergeFrom := fbParseCtx.ReadUint32(anyUdint:= _stDevice.id); 
    16#1A:    // repeated uint32 error_codes = 3;
        MergeFrom := _fbRepeatedId3.AddEntriesFrom(fbParseCtx:= fbParseCtx, ipFieldCodec:= _fbFieldCodecId3,nCount=> _stDevice.error_codes_count);
    16#20:    // int32 temperature = 4;
        MergeFrom := fbParseCtx.ReadInt32(anyDint:= _stDevice.temperature); 
    16#2A:    // bytes data = 5;
        MergeFrom := fbParseCtx.ReadBytes(aBytes:= _stDevice.data, nCount=> _stDevice.data_count); 
ELSE
    MergeFrom := fbParseCtx.SkipLastField();
END_CASE

UNTIL (FAILED(MergeFrom) OR nTag = 0)
END_REPEAT
END_METHOD

PROPERTY PUBLIC MessageValue : T_Any
GET
MessageValue := F_ToAnyType(anyArg:= _stDevice);
END_GET
END_PROPERTY

PROPERTY PUBLIC Parser : REFERENCE TO FB_MessageParser
GET
Parser REF= THIS^._fbMessageParser;
END_GET
END_PROPERTY

(* Writer for this message.*)
PROPERTY PUBLIC Writer : REFERENCE TO FB_MessageWriter
GET
Writer REF= THIS^._fbMessageWriter;
END_GET
END_PROPERTY

(* Writes the data to the given coded output stream.*)
{attribute 'no-analysis'}
METHOD WriteTo : HRESULT
VAR_IN_OUT
	(* Coded output stream to write the data to. *)
	fbWriteCtx	: FB_WriteContext;
END_VAR
// string name = 1;
WriteTo := fbWriteCtx.WriteTag(1, E_WireType.LengthDelimited);
IF FAILED(WriteTo) THEN
    RETURN;
END_IF
WriteTo := fbWriteCtx.WriteString(sStringToWrite:= _stDevice.name);
IF FAILED(WriteTo) THEN
    RETURN;
END_IF
// uint32 id = 2;
WriteTo := fbWriteCtx.WriteTag(2, E_WireType.Varint);
IF FAILED(WriteTo) THEN
    RETURN;
END_IF
WriteTo := fbWriteCtx.WriteUint32(anyUdint:= _stDevice.id);
IF FAILED(WriteTo) THEN
    RETURN;
END_IF
// repeated uint32 error_codes = 3;
WriteTo := _fbRepeatedId3.WriteToWithCount(fbWriteCtx:= fbWriteCtx, ipFieldCodec:= _fbFieldCodecId3, nCount:= _stDevice.error_codes_count);
IF FAILED(WriteTo) THEN
    RETURN;
END_IF
// int32 temperature = 4;
WriteTo := fbWriteCtx.WriteTag(4, E_WireType.Varint);
IF FAILED(WriteTo) THEN
    RETURN;
END_IF
WriteTo := fbWriteCtx.WriteInt32(anyDint:= _stDevice.temperature);
IF FAILED(WriteTo) THEN
    RETURN;
END_IF
// bytes data = 5;
WriteTo := fbWriteCtx.WriteTag(5, E_WireType.LengthDelimited);
IF FAILED(WriteTo) THEN
    RETURN;
END_IF
WriteTo := fbWriteCtx.WriteBytes(aBytes:= _stDevice.data, nCount:= _stDevice.data_count);
IF FAILED(WriteTo) THEN
    RETURN;
END_IF
END_METHOD

END_FUNCTION_BLOCK

// ---- __TESTs/WireFormatTests/PRG_WireFormatTests.TcPOU
{attribute 'analysis' := '-33'}
PROGRAM INTERNAL PRG_WireFormatTests
{IF defined (UNIT_TEST)}
    fbMakeTagTests       : FB_MakeTagTests;
{END_IF}

END_PROGRAM

// ---- __TESTs/WireFormatTests/FB_MakeTagTests.TcPOU
FUNCTION_BLOCK INTERNAL FINAL FB_MakeTagTests EXTENDS FB_TestSuite
VAR_INPUT
END_VAR
VAR_OUTPUT
END_VAR
VAR
    nActualTag : UDINT;
END_VAR

TEST(__POUNAME());

// Arrange

// Act
nActualTag := F_MakeTag(nFieldNumber:= 6, eWireType:= E_WireType.LengthDelimited);

// Assert
AssertEquals_UDINT(Expected:= 16#32, Actual:= nActualTag, Message:= '');


TEST_FINISHED_NAMED(__POUNAME());

END_FUNCTION_BLOCK

// ---- WireFormat/POus/F_MakeTag.TcPOU
// Makes a tag value given a field number and wire type.
FUNCTION F_MakeTag : UDINT
VAR_INPUT
    nFieldNumber    : UDINT;
    eWireType       : E_WireType;
END_VAR
VAR
END_VAR


F_MakeTag := SHL(nFieldNumber, GCL_WireFormat.cTagTypeBits) OR eWireType;

END_FUNCTION

// ---- __TESTs/EnumTests/PRG_EnumTests.TcPOU
{attribute 'analysis' := '-33'}
PROGRAM INTERNAL PRG_EnumTests
VAR
{IF defined (UNIT_TEST)}
	fbF_ComputeEnumSizeTests : FB_F_ComputeEnumSizeTests;
{END_IF}
END_VAR

END_PROGRAM

// ---- __TESTs/EnumTests/FB_F_ComputeEnumSizeTests.TcPOU
FUNCTION_BLOCK INTERNAL FINAL FB_F_ComputeEnumSizeTests EXTENDS FB_TestSuite
VAR_INPUT
END_VAR
VAR_OUTPUT
END_VAR
VAR
	aValues	: ARRAY[0..5] OF E_INT := [E_INT.eVAL0, E_INT.eVAL1, E_INT.eVAL2, E_INT.eVAL3, E_INT.eMIN, E_INT.eMAX];
	nActual : UDINT;
	i : UDINT;
END_VAR

TEST(__POUNAME());

//Arrange
nActual := 0;

// Act
FOR i := 0  TO 5 DO
    nActual := nActual + F_ComputeEnumSize(anyEnum:= aValues[i]);
END_FOR

//Assert
AssertEquals_UDINT(Expected:= 10, Actual:= nActual, Message:= '');

TEST_FINISHED_NAMED(__POUNAME());

END_FUNCTION_BLOCK

// ---- __TESTs/RepeatedFieldTests/PRG_RepeatedFieldTests.TcPOU
{attribute 'analysis' := '-33'}
PROGRAM INTERNAL PRG_RepeatedFieldTests
{IF defined (UNIT_TEST)}

{END_IF}

PRG_ReadRepeatedFieldTests();
PRG_WriteRepeatedFieldTests();
PRG_RoundTripRepeatedFieldTests();

END_PROGRAM

// ---- __TESTs/RepeatedFieldTests/Read/PRG_ReadRepeatedFieldTests.TcPOU
{attribute 'analysis' := '-33'}
PROGRAM INTERNAL PRG_ReadRepeatedFieldTests
{IF defined (UNIT_TEST)}
	fbReadRepeatedFieldBoolTests    : FB_ReadRepeatedFieldBoolTests;
	fbReadRepeatedFieldBytesTests   : FB_ReadRepeatedFieldBytesTests;
	fbReadRepeatedFieldEnumTests 	: FB_ReadRepeatedFieldEnumTests;
    fbReadRepeatedFieldUint32Tests  : FB_ReadRepeatedFieldUint32Tests;
    fbReadRepeatedFieldFixed32Tests : FB_ReadRepeatedFieldFixed32Tests;
    fbReadRepeatedFieldFixed64Tests : FB_ReadRepeatedFieldFixed64Tests;
    fbReadRepeatedFieldStringTests  : FB_ReadRepeatedFieldStringTests;
{END_IF}

END_PROGRAM

// ---- __TESTs/RepeatedFieldTests/Read/FB_ReadRepeatedFieldBoolTests.TcPOU
FUNCTION_BLOCK INTERNAL FINAL FB_ReadRepeatedFieldBoolTests EXTENDS FB_TestSuite
VAR_INPUT
END_VAR
VAR_OUTPUT
END_VAR
VAR
	aActual             : ARRAY [0..15] OF BOOL;
    fbFieldCodec 		: FB_FieldCodecBool(nTag:= 16#0A);
	fbRepeatedField		: FB_RepeatedField(anyArray:= F_ToAnyType(aActual), anyFirstElem:= F_ToAnyType(aActual[0]), ipFieldCodec:= fbFieldCodec);
END_VAR

ShouldReadRepeatedFieldTheory();

METHOD PRIVATE Reset
VAR_INPUT
END_VAR
fbRepeatedField.Initialize();
MEMSET(destAddr:= ADR(aActual), fillByte:= 16#0, n:= SIZEOF(aActual));
END_METHOD

METHOD PRIVATE ShouldReadRepeatedField
VAR_IN_OUT CONSTANT
    aBuffer     : ARRAY [*] OF BYTE;
    aExpected   : ARRAY [*] OF BOOL;
END_VAR
VAR_INPUT CONSTANT
    nBufferPosStart     : UDINT;
    nExpectedBufferPos  : UDINT;
    nExpectedFieldIndex : UDINT;
    ipFieldCodec        : I_FieldCodec;
END_VAR
VAR_INST
    fbCtx               : FB_ParseContext;
END_VAR
VAR    
    hr                  : HRESULT;
    nTag                : UDINT;
END_VAR
// Arrange
Reset();
fbCtx.FromBuffer(aBuffer);
fbCtx.refCtx.stState.nBufferPos := nBufferPosStart;

// Act
F_ParseTag(fbCtx.refCtx, nTag=> nTag);
hr := fbRepeatedField.AddEntriesFrom(fbParseCtx:= fbCtx, ipFieldCodec:= ipFieldCodec);

// Assert
AssertEquals_DINT(
    Expected:= S_OK,
    Actual:= hr,
    Message:= 'Expected S_OK instead of error');
    
{warning disable C0041}
AssertArrayEquals_BOOL(Expecteds:= aExpected, Actuals:= aActual, Message:= '');
 
AssertEquals_UDINT(
    Expected:= nExpectedBufferPos,
    Actual:= fbCtx.refCtx.stState.nBufferPos,
    Message:= CONCAT('Expected stState.nBufferPos to equal ', TO_STRING(nExpectedBufferPos)));
    
AssertEquals_UDINT(
    Expected:= nExpectedFieldIndex,
    Actual:= fbRepeatedField.nCount,
    Message:= CONCAT('Expected fbRepeatedField.nCount to equal ', TO_STRING(nExpectedFieldIndex)));
END_METHOD

METHOD PRIVATE ShouldReadRepeatedFieldTheory : REFERENCE TO FB_Test
VAR CONSTANT
    cRawValueZeroLength     : ARRAY[0..15] OF BYTE := [16#0A, 16#00];
    cRawValue1              : ARRAY[0..15] OF BYTE := [16#00, 16#0A, 16#05, 16#01, 16#00, 16#01, 16#01, 16#00];
END_VAR

VAR CONSTANT
    aExpectedZeroLength     : ARRAY [0..15] OF BOOL := [0, 0, 0, 0, 0, 0, 0, 0, 0, 0, 0, 0, 0, 0, 0, 0];
    aExpected1              : ARRAY [0..15] OF BOOL := [TRUE, FALSE, TRUE, TRUE, FALSE];
END_VAR
TEST(__POUNAME());

ShouldReadRepeatedField(aBuffer:= cRawValueZeroLength, aExpected:= aExpectedZeroLength, nBufferPosStart:= 0, nExpectedBufferPos:= 2, nExpectedFieldIndex:= 0, ipFieldCodec:= THIS^.fbFieldCodec);
ShouldReadRepeatedField(aBuffer:= cRawValue1, aExpected:= aExpected1, nBufferPosStart:= 1, nExpectedBufferPos:= 8, nExpectedFieldIndex:= 5, ipFieldCodec:= THIS^.fbFieldCodec);

TEST_FINISHED_NAMED(__POUNAME());
END_METHOD

END_FUNCTION_BLOCK

// ---- FieldCodec/FB_FieldCodecBool.TcPOU
FUNCTION_BLOCK FB_FieldCodecBool EXTENDS FB_FieldCodec
VAR_INPUT
END_VAR
VAR_OUTPUT
END_VAR
VAR
    bValue : BOOL;
END_VAR

METHOD CalculatePackedDataSize : HRESULT
VAR_INPUT CONSTANT
	anyFirstElem	: T_Any;
	nLength	        : UDINT;        // items to write
END_VAR
VAR_OUTPUT
    nPackedDataSize : UDINT;
END_VAR
VAR
    anyItem         : T_ANY;
    i               : UDINT;
    nValue          : BYTE;
END_VAR
anyItem := anyFirstElem;

IF nLength < 1 THEN
    nPackedDataSize := 0;
    RETURN;
END_IF

FOR i := 0  TO nLength - 1 DO
    anyItem.pValue := anyFirstElem.pValue + (i * TO_UDINT(anyFirstElem.diSize)); 
    nValue := PBYTE_TO_BYTE(anyItem.pValue);
    nPackedDataSize := nPackedDataSize + GCL_PB.cBoolSize;
END_FOR
END_METHOD

METHOD IsPackedRepeatedField : BOOL
VAR_INPUT
	nTag	: UDINT;
END_VAR
IsPackedRepeatedField := F_IsPackedRepeatedField(nTag);
END_METHOD


METHOD ValueReader : HRESULT
VAR_IN_OUT
    stCtx : ST_ParseContext;
END_VAR
VAR_OUTPUT
	anyOut	: T_Any;
END_VAR

ValueReader := F_ParseRawVarint32(stCtx, bValue);
anyOut := F_ToAnyType(anyArg:= bValue);
END_METHOD

METHOD ValueWriter : HRESULT
VAR_IN_OUT
    stCtx  : ST_WriteContext;
END_VAR
VAR_INPUT
    anyIn : T_ANY;
END_VAR
VAR
	nValue : BYTE;
END_VAR

nValue := PBYTE_TO_BYTE(anyIn.pValue);
ValueWriter := F_WriteRawByte(stCtx, nValue);
END_METHOD

END_FUNCTION_BLOCK

// ---- __TESTs/RepeatedFieldTests/Read/FB_ReadRepeatedFieldBytesTests.TcPOU
FUNCTION_BLOCK INTERNAL FINAL FB_ReadRepeatedFieldBytesTests EXTENDS FB_TestSuite
VAR_INPUT
END_VAR
VAR_OUTPUT
END_VAR
VAR
	aActual             : ARRAY[0..3] OF ARRAY[0..15] OF BYTE;
    fbFieldCodec 		: FB_FieldCodecBytes(nTag:= 16#22);
	fbRepeatedField		: FB_RepeatedField(anyArray:= F_ToAnyType(aActual), anyFirstElem:= F_ToAnyType(aActual[0]), ipFieldCodec:= fbFieldCodec);
END_VAR

ShouldReadRepeatedFieldTheory();

METHOD PRIVATE Reset
VAR_INPUT
END_VAR
fbRepeatedField.Initialize();
MEMSET(destAddr:= ADR(aActual), fillByte:= 16#0, n:= SIZEOF(aActual));
END_METHOD

METHOD PRIVATE ShouldReadRepeatedField
VAR_IN_OUT CONSTANT
    aBuffer     : ARRAY [*] OF BYTE;
    aExpected   : ARRAY[0..3] OF ARRAY[0..15] OF BYTE;
END_VAR
VAR_INPUT CONSTANT
    nBufferPosStart     : UDINT;
    nExpectedBufferPos  : UDINT;
    nExpectedFieldIndex : UDINT;
    ipFieldCodec        : I_FieldCodec;
END_VAR
VAR_INST
    fbCtx               : FB_ParseContext;
END_VAR
VAR
    hr                  : HRESULT;
    nTag                : UDINT;
    i                   : UDINT;
    aTmpBuffer          : ARRAY[0..1023] OF BYTE := [SIZEOF(aTmpBuffer)(16#FF)];
END_VAR
// Arrange
Reset();
fbCtx.FromBuffer(aBuffer);
fbCtx.refCtx.stState.nBufferPos := nBufferPosStart;
THIS^.fbFieldCodec.SetTmpBuffer(anyBytes:= F_ToAnyBytes(aTmpBuffer));

// Act
F_ParseTag(fbCtx.refCtx, nTag=> nTag);
hr := fbRepeatedField.AddEntriesFrom(fbParseCtx:= fbCtx, ipFieldCodec:= ipFieldCodec);

// Assert
AssertEquals_DINT(
    Expected:= S_OK,
    Actual:= hr,
    Message:= 'Expected S_OK instead of error');
    
{warning disable C0041}
FOR i:= 0 TO 3 DO
    AssertArrayEquals_BYTE(Expecteds:= aExpected[i], Actuals:= aActual[i], Message:= CONCAT('Array differs at index ', TO_STRING(i)));
END_FOR

AssertEquals_UDINT(
    Expected:= nExpectedBufferPos,
    Actual:= fbCtx.refCtx.stState.nBufferPos,
    Message:= CONCAT('Expected stState.nBufferPos to equal ', TO_STRING(nExpectedBufferPos)));
    
AssertEquals_UDINT(
    Expected:= nExpectedFieldIndex,
    Actual:= fbRepeatedField.nCount,
    Message:= CONCAT('Expected fbRepeatedField.nCount to equal ', TO_STRING(fbRepeatedField.nCount)));
END_METHOD

METHOD PRIVATE ShouldReadRepeatedFieldTheory : REFERENCE TO FB_Test
(*
    syntax = "proto3";
    
    message exampleMessage
    {
      repeated bytes repeatedBytes = 4;
    }    
*)

VAR CONSTANT
    cRawBytes1 : ARRAY[0..31] OF BYTE := [16#22, 16#03, 16#00, 16#01, 16#02, 16#22, 16#03, 16#03, 16#04, 16#05];
    
END_VAR

VAR CONSTANT
     aExpected1 : ARRAY[0..3] OF ARRAY[0..15] OF BYTE := [[0, 1, 2], [3, 4, 5]];
END_VAR
VAR
    // aBuffer     : ARRAY[0..1023] OF BYTE;       // tmp. buffer if chunks are larger then 256 bytes.
END_VAR
TEST(__POUNAME());

ShouldReadRepeatedField(aBuffer:= cRawBytes1, aExpected:= aExpected1, nBufferPosStart:= 0, nExpectedBufferPos:= 11, nExpectedFieldIndex:= 2, THIS^.fbFieldCodec);

TEST_FINISHED_NAMED(__POUNAME());
END_METHOD

END_FUNCTION_BLOCK

// ---- FieldCodec/FB_FieldCodecBytes.TcPOU
FUNCTION_BLOCK FB_FieldCodecBytes Extends FB_FieldCodec
VAR_INPUT
END_VAR
VAR_OUTPUT
END_VAR
VAR
    aValue      : ARRAY[0..Param_PB.cFieldCodecBytesDefaultSize - 1] OF BYTE;        // default buffer size, if more bytes are needed, set size with "SetAnyBytes" method.
    tAnyBytes : T_AnyBytes;
END_VAR

{attribute 'analysis' := '-33'}
METHOD CalculatePackedDataSize : HRESULT
VAR_INPUT CONSTANT
	anyFirstElem	: T_Any;
	nLength	        : UDINT;        // items to write
END_VAR
VAR_OUTPUT
    nPackedDataSize : UDINT;
END_VAR

CalculatePackedDataSize := 0;
END_METHOD

METHOD IsPackedRepeatedField : BOOL
VAR_INPUT
    {attribute 'analysis' := '-33' } 
	nTag	: UDINT;
END_VAR

IsPackedRepeatedField := FALSE;
END_METHOD

// Map ARRAY [*] OF BYTE for field repeated bytes
METHOD INTERNAL SetTmpBuffer
VAR_INPUT
    anyBytes : T_AnyBytes;
END_VAR
THIS^.tAnyBytes := anyBytes;
END_METHOD


METHOD ValueReader : HRESULT
VAR_IN_OUT      
    stCtx : ST_ParseContext;
END_VAR
VAR_OUTPUT
	anyOut	: T_Any;
END_VAR
VAR
    nLength : UDINT;
END_VAR

ValueReader := F_ParseLength(stCtx, nLength=> nLength);
IF FAILED(ValueReader) THEN
    RETURN;
END_IF

IF tAnyBytes.pValue <> NULL THEN
    anyOut := tAnyBytes;
ELSE
    anyOut := F_ToAnyBytes(aValue);
END_IF

ValueReader := F_ReadRawBytes(stCtx, anyOut, nLength);
anyOut.diSize := TO_DINT(nLength);
END_METHOD

METHOD ValueWriter : HRESULT
VAR_IN_OUT
    stCtx  : ST_WriteContext;
END_VAR
VAR_INPUT
    anyIn : T_ANY;
END_VAR
{warning 'FIXME: This should write the actual number of bytes, otherwise we waste space on the wire...'}
ValueWriter := F_WriteLength(stCtx, TO_UDINT(anyin.diSize));
IF SUCCEEDED(ValueWriter) THEN
	ValueWriter := F_WriteRawBytes(stCtx, anyIn, TO_UDINT(anyin.diSize));
END_IF
END_METHOD

END_FUNCTION_BLOCK

// ---- __TESTs/RepeatedFieldTests/Read/FB_ReadRepeatedFieldEnumTests.TcPOU
FUNCTION_BLOCK  INTERNAL FINAL FB_ReadRepeatedFieldEnumTests EXTENDS FB_TestSuite
VAR_INPUT
END_VAR
VAR_OUTPUT
END_VAR
VAR
	fbSUT : FB_FieldCodecEnum(nTag:= 16#0A);
END_VAR

ShouldReadEnumWithBaseTypeByte();
ShouldReadEnumWithBaseTypeInt();

METHOD PRIVATE ShouldReadEnumWithBaseTypeByte : HRESULT
{region 'proto'} (*
syntax = "proto3";
import "tchaxx-extensions.proto";
message FieldCodecEnumTests {
  enum ByteEnum {
	option (tchaxx.enum_integer_type) = EIT_BYTE;
    MIN = 0;
    VAL1 = 1;
    VAL2 = 2;
    VAL3 = 3;
    MAX = 255;
  }
  repeated ByteEnum byte_enum = 1 [(tchaxx.array_len) = 8;
}
*){endregion}

VAR
	aActualValues : ARRAY[0..7] OF E_BYTE;
	aExpectedValues : ARRAY[0..7] OF E_BYTE := [E_BYTE.eMIN, E_BYTE.eMAX, E_BYTE.eVAL3, E_BYTE.eVAL2, E_BYTE.eVAL1, E_BYTE.eVAL2, E_BYTE.eVAL3];
	fbCtx : FB_ParseContext;
	fbRepeatedField	: FB_RepeatedField(anyArray:= F_ToAnyType(aActualValues), anyFirstElem:= F_ToAnyType(aActualValues[0]), ipFieldCodec:= fbSUT);
END_VAR
VAR CONSTANT
	// 0a0900ff01030201820203 -> decoded "byte_enum": [ "MIN", "MAX", "VAL3", "VAL2", "VAL1", 258, "VAL3" ] where 258 should overflow to "VAL2"
	cBuffer : ARRAY[0..63] OF BYTE := [16#0A, 16#09, 16#00, 16#FF, 16#01, 16#03, 16#02, 16#01, 16#82, 16#02, 16#03];
	cExpectedBufferPos : UDINT := 11;
	cExpectedFieldIndex : UDINT := 7;
END_VAR
VAR
	nTag : UDINT;
	hr : HRESULT;
END_VAR
TEST(__POUNAME());

// Arrange
fbCtx.FromBuffer(cBuffer);

// Act
F_ParseTag(fbCtx.refCtx, nTag=> nTag);
hr := fbRepeatedField.AddEntriesFrom(fbParseCtx:= fbCtx, ipFieldCodec:= fbSUT);

// Assert
AssertEquals_DINT(
    Expected:= S_OK,
    Actual:= hr,
    Message:= 'Expected S_OK instead of error');
	
AssertEquals(Expected:= aExpectedValues, Actual:= aActualValues, Message:= '');
AssertEquals_UDINT(
    Expected:= cExpectedBufferPos,
    Actual:= fbCtx.refCtx.stState.nBufferPos,
    Message:= CONCAT('Expected stState.nBufferPos to equal ', TO_STRING(cExpectedBufferPos)));
    
AssertEquals_UDINT(
    Expected:= cExpectedFieldIndex,
    Actual:= fbRepeatedField.nCount,
    Message:= CONCAT('Expected fbRepeatedField.nCount to equal ', TO_STRING(cExpectedFieldIndex)));
	
TEST_FINISHED_NAMED(__POUNAME());
END_METHOD

METHOD PRIVATE ShouldReadEnumWithBaseTypeInt : HRESULT
{region 'proto'} (*
syntax = "proto3";
import "tchaxx-extensions.proto";
message FieldCodecEnumTests {
  enum IntEnum {
	option (tchaxx.enum_integer_type) = EIT_INT;
    VAL0 = 0;
    MIN = -32768;
    VAL1 = 1;
    VAL2 = 2;
    VAL3 = 3;
    MAX = 32767;
  }
  repeated IntEnum int_enum = 1 [(tchaxx.array_len) = 8];
}
*){endregion}

VAR	
	aActualValues : ARRAY[0..7] OF E_INT;
	aExpectedValues : ARRAY[0..7] OF E_INT := [E_INT.eVAL0, E_INT.eMIN, E_INT.eMAX, E_INT.eVAL3, E_INT.eVAL2, E_INT.eVAL1];
	fbCtx : FB_ParseContext;
	fbRepeatedField	: FB_RepeatedField(anyArray:= F_ToAnyType(aActualValues), anyFirstElem:= F_ToAnyType(aActualValues[0]), ipFieldCodec:= fbSUT);
END_VAR
VAR CONSTANT
	// 0a11008080feffffffffffff01ffff01030201 -> decoded "byte_enum": [ "VAL0", "MIN", "MAX", "VAL3", "VAL2", "VAL1"]
	cBuffer : ARRAY[0..63] OF BYTE := [16#0A, 16#11, 16#00, 16#80, 16#80, 16#FE, 16#FF, 16#FF, 16#FF, 16#FF, 16#FF, 16#FF, 16#01, 16#FF, 16#FF, 16#01, 16#03, 16#02, 16#01];
	cExpectedBufferPos : UDINT := 19;
	cExpectedFieldIndex : UDINT := 6;
END_VAR
VAR
	nTag : UDINT;
	hr : HRESULT;
END_VAR
TEST(__POUNAME());

// Arrange
fbCtx.FromBuffer(cBuffer);

// Act
F_ParseTag(fbCtx.refCtx, nTag=> nTag);
hr := fbRepeatedField.AddEntriesFrom(fbParseCtx:= fbCtx, ipFieldCodec:= fbSUT);

// Assert
AssertEquals_DINT(
    Expected:= S_OK,
    Actual:= hr,
    Message:= 'Expected S_OK instead of error');
	
AssertEquals(Expected:= aExpectedValues, Actual:= aActualValues, Message:= '');
AssertEquals_UDINT(
    Expected:= cExpectedBufferPos,
    Actual:= fbCtx.refCtx.stState.nBufferPos,
    Message:= CONCAT('Expected stState.nBufferPos to equal ', TO_STRING(cExpectedBufferPos)));
    
AssertEquals_UDINT(
    Expected:= cExpectedFieldIndex,
    Actual:= fbRepeatedField.nCount,
    Message:= CONCAT('Expected fbRepeatedField.nCount to equal ', TO_STRING(cExpectedFieldIndex)));
	
TEST_FINISHED_NAMED(__POUNAME());
END_METHOD

END_FUNCTION_BLOCK

// ---- FieldCodec/FB_FieldCodecEnum.TcPOU
FUNCTION_BLOCK FB_FieldCodecEnum EXTENDS FB_FieldCodec
VAR_INPUT
END_VAR
VAR_OUTPUT
END_VAR
VAR
	nValue : DINT;
END_VAR

METHOD CalculatePackedDataSize : HRESULT
VAR_INPUT CONSTANT
	anyFirstElem	: T_Any;
	nLength	        : UDINT;        // items to write
END_VAR
VAR_OUTPUT
    nPackedDataSize : UDINT;
END_VAR
VAR
    anyItem         : T_ANY;
    i               : UDINT;
END_VAR
IF anyFirstElem.pValue = NULL OR anyFirstElem.TypeClass <> __SYSTEM.TYPE_CLASS.TYPE_ENUM THEN
    CalculatePackedDataSize := E_HRESULTAdsErr.INVALIDDATA;
    RETURN;
END_IF

anyItem := anyFirstElem;

IF nLength < 1 THEN
    nPackedDataSize := 0;
    RETURN;
END_IF

FOR i := 0  TO nLength - 1 DO
    anyItem.pValue := anyFirstElem.pValue + (i * TO_UDINT(anyFirstElem.diSize)); 
    nPackedDataSize := nPackedDataSize + F_ComputeEnumSize(anyItem);
END_FOR
END_METHOD

METHOD IsPackedRepeatedField : BOOL
VAR_INPUT
	nTag	: UDINT;
END_VAR
IsPackedRepeatedField := F_IsPackedRepeatedField(nTag);
END_METHOD


METHOD ValueReader : HRESULT
VAR_IN_OUT      
    stCtx : ST_ParseContext;
END_VAR
VAR_OUTPUT
	anyOut	: T_Any;
END_VAR

ValueReader := F_ParseRawVarint32(stCtx, nValue);
IF FAILED(ValueReader) THEN
    RETURN;
END_IF
anyOut := F_ToAnyType(anyArg:= nValue);
END_METHOD

METHOD ValueWriter : HRESULT
VAR_IN_OUT
    stCtx  : ST_WriteContext;
END_VAR
VAR_INPUT
    anyIn : T_ANY;
END_VAR
VAR
    nValue  : DINT;
END_VAR
IF anyIn.pValue = NULL OR anyIn.TypeClass <> __SYSTEM.TYPE_CLASS.TYPE_ENUM THEN
    ValueWriter := E_HRESULTAdsErr.INVALIDDATA;
    RETURN;
END_IF

MEMCPY(destAddr:= ADR(nValue), srcAddr:= anyIn.pValue, MIN(TO_UDINT(anyIn.diSize), SIZEOF(nValue)));
ValueWriter := F_WriteInt32(stCtx, nValue);
END_METHOD

END_FUNCTION_BLOCK

// ---- __TESTs/RepeatedFieldTests/Read/FB_ReadRepeatedFieldUint32Tests.TcPOU
FUNCTION_BLOCK INTERNAL FINAL FB_ReadRepeatedFieldUint32Tests EXTENDS FB_TestSuite
VAR_INPUT
END_VAR
VAR_OUTPUT
END_VAR
VAR
	aActual             : ARRAY [0..15] OF UDINT;
	fbFieldCodec 		: FB_FieldCodecUInt32(nTag:= 16#0A);
	fbRepeatedField		: FB_RepeatedField(anyArray:= F_ToAnyType(aActual), anyFirstElem:= F_ToAnyType(aActual[0]), ipFieldCodec:= fbFieldCodec);
END_VAR

ShouldReadRepeatedFieldTheory();
ShouldReadNonConsecutiveRepeatedFields();

METHOD PRIVATE Reset
VAR_INPUT
END_VAR
fbRepeatedField.Initialize();
MEMSET(destAddr:= ADR(aActual), fillByte:= 16#0, n:= SIZEOF(aActual));
END_METHOD

METHOD PRIVATE ShouldReadNonConsecutiveRepeatedFields
VAR CONSTANT
    (*
        message Demo {
            repeated uint32 a = 1;
            fixed32 b =2;
        }
        JSON:
        {
          "a": [
            0, 1, 2, 151
          ],
          "b": 321
        }
    *)
    cRawMessage : ARRAY[0..15] OF BYTE := [16#0A, 16#03, 16#00, 16#01, 16#02, 16#15, 16#41, 16#01, 16#00, 16#00, 16#0A, 16#02, 16#97, 16#01];
    cExpected   : ARRAY[0..15] OF UDINT := [0, 1, 2, 151];
END_VAR
VAR_INST
    fbCtx               : FB_ParseContext;
END_VAR
VAR
    hr                  : HRESULT;
    nB                  : UDINT;
END_VAR
TEST(__POUNAME());

// Arrange
Reset();
fbCtx.FromBuffer(cRawMessage);

// Act
// Parses a=[0,1,2]: 16#0A, 16#03, 16#00, 16#01, 16#02
F_ParseTag(fbCtx.refCtx, nTag=> );
hr := fbRepeatedField.AddEntriesFrom(fbParseCtx:= fbCtx, ipFieldCodec:= fbFieldCodec);

// Parses b=321: 16#15, 16#41, 16#01, 16#00, 16#00
F_ParseTag(fbCtx.refCtx, nTag=> );
F_ParseRawLittleEndian32(fbCtx.refCtx, nValue=> nB);

// Parses a=[151]: 16#0A, 16#02, 16#97, 16#01
F_ParseTag(fbCtx.refCtx, nTag=> );
hr := fbRepeatedField.AddEntriesFrom(fbParseCtx:= fbCtx, ipFieldCodec:= fbFieldCodec);

// Assert
AssertEquals_DINT(
    Expected:= S_OK,
    Actual:= hr,
    Message:= 'Expected S_OK instead of error');
    
{warning disable C0041}
AssertArrayEquals_UDINT(Expecteds:= cExpected, Actuals:= aActual, Message:= '');
    
AssertEquals_UDINT(
    Expected:= 4,
    Actual:= fbRepeatedField.nCount,
    Message:= CONCAT('Expected fbRepeatedField.nCount to equal ', TO_STRING(4)));
   
AssertEquals_UDINT(
    Expected:= 321,
    Actual:= nB,
    Message:= CONCAT('Expected nB to equal ', TO_STRING(321)));
 
TEST_FINISHED_NAMED(__POUNAME());
END_METHOD

METHOD PRIVATE ShouldReadRepeatedField
VAR_IN_OUT CONSTANT
    aBuffer   			: ARRAY [*] OF BYTE;
    aExpected 			: ARRAY [*] OF UDINT;
END_VAR
VAR_INPUT CONSTANT
    nBufferPosStart     : UDINT;
    nExpectedBufferPos  : UDINT;
    nExpectedFieldIndex : UDINT;
    ipFieldCodec        : I_FieldCodec;
END_VAR
VAR_INST
    fbCtx               : FB_ParseContext;
END_VAR
VAR    
    hr                  : HRESULT;
    nTag                : UDINT;
END_VAR
// Arrange
Reset();
fbCtx.FromBuffer(aBuffer);
fbCtx.refCtx.stState.nBufferPos := nBufferPosStart;

// Act
F_ParseTag(fbCtx.refCtx, nTag=> nTag);
hr := fbRepeatedField.AddEntriesFrom(fbParseCtx:= fbCtx, ipFieldCodec:= ipFieldCodec);

// Assert
AssertEquals_DINT(
    Expected:= S_OK,
    Actual:= hr,
    Message:= 'Expected S_OK instead of error');
    
{warning disable C0041}
AssertArrayEquals_UDINT(Expecteds:= aExpected, Actuals:= aActual, Message:= '');
 
AssertEquals_UDINT(
    Expected:= nExpectedBufferPos,
    Actual:= fbCtx.refCtx.stState.nBufferPos,
    Message:= CONCAT('Expected stState.nBufferPos to equal ', TO_STRING(nExpectedBufferPos)));
    
AssertEquals_UDINT(
    Expected:= nExpectedFieldIndex,
    Actual:= fbRepeatedField.nCount,
    Message:= CONCAT('Expected fbRepeatedField.nCount to equal ', TO_STRING(nExpectedFieldIndex)));
END_METHOD

{warning 'TODO: Add better tests for UInt32'}
METHOD PRIVATE ShouldReadRepeatedFieldTheory : REFERENCE TO FB_Test
VAR CONSTANT
    cRawValueZeroLength     : ARRAY[0..15] OF BYTE := [16#0A, 16#00];
    cRawValue1              : ARRAY[0..15] OF BYTE := [16#00, 16#0A, 16#07, 16#00, 16#01, 16#FF, 16#01, 16#96, 16#01, 16#04];
END_VAR

VAR CONSTANT
    aExpectedZeroLength     : ARRAY [0..15] OF UDINT := [0, 0, 0, 0, 0, 0, 0, 0, 0, 0, 0, 0, 0, 0, 0, 0];
    aExpected1             	: ARRAY [0..15] OF UDINT := [0, 1, 255, 150, 4, 0, 0, 0, 0, 0, 0, 0, 0, 0, 0, 0];
END_VAR
TEST(__POUNAME());

ShouldReadRepeatedField(aBuffer:= cRawValueZeroLength, aExpected:= aExpectedZeroLength, nBufferPosStart:= 0, nExpectedBufferPos:= 2, nExpectedFieldIndex:= 0, ipFieldCodec:= THIS^.fbFieldCodec);
ShouldReadRepeatedField(aBuffer:= cRawValue1, aExpected:= aExpected1, nBufferPosStart:= 1, nExpectedBufferPos:= 10, nExpectedFieldIndex:= 5, ipFieldCodec:= THIS^.fbFieldCodec);

TEST_FINISHED_NAMED(__POUNAME());
END_METHOD

END_FUNCTION_BLOCK

// ---- __TESTs/RepeatedFieldTests/Read/FB_ReadRepeatedFieldFixed32Tests.TcPOU
FUNCTION_BLOCK INTERNAL FINAL FB_ReadRepeatedFieldFixed32Tests EXTENDS FB_TestSuite
VAR_INPUT
END_VAR
VAR_OUTPUT
END_VAR
VAR
	aActual             : ARRAY [0..7] OF DINT;
	fbFieldCodec 		: FB_FieldCodecFixed32(nTag:= 16#0A);
	fbRepeatedField	: FB_RepeatedField(anyArray:= F_ToAnyType(aActual), anyFirstElem:= F_ToAnyType(aActual[0]), ipFieldCodec:= fbFieldCodec);
END_VAR

ShouldReadRepeatedFieldTheory();

METHOD PRIVATE Reset
VAR_INPUT
END_VAR
fbRepeatedField.Initialize();
MEMSET(destAddr:= ADR(aActual), fillByte:= 16#0, n:= SIZEOF(aActual[0]));
END_METHOD

METHOD PRIVATE ShouldReadRepeatedField
VAR_IN_OUT CONSTANT
    aBuffer     : ARRAY [*] OF BYTE;
    aExpected   : ARRAY [*] OF DINT;
END_VAR
VAR_INPUT CONSTANT
    nBufferPosStart     : UDINT;
    nExpectedBufferPos  : UDINT;
    nExpectedFieldIndex : UDINT;
    ipFieldCodec        : I_FieldCodec;
END_VAR
VAR_INST
    fbCtx               : FB_ParseContext;
END_VAR
VAR
    hr                  : HRESULT;
	nTag                : UDINT;
END_VAR
// Arrange
Reset();
fbCtx.FromBuffer(aBuffer);
fbCtx.refCtx.stState.nBufferPos := nBufferPosStart;;

// Act
F_ParseTag(fbCtx.refCtx, nTag=> nTag);
hr := fbRepeatedField.AddEntriesFrom(fbParseCtx:= fbCtx, ipFieldCodec:= ipFieldCodec);

// Assert
AssertEquals_DINT(
    Expected:= S_OK,
    Actual:= hr,
    Message:= 'Expected S_OK instead of error');
    
{warning disable C0041}
AssertArrayEquals_DINT(Expecteds:= aExpected, Actuals:= aActual, Message:= '');
 
AssertEquals_UDINT(
    Expected:= nExpectedBufferPos,
    Actual:= fbCtx.refCtx.stState.nBufferPos,
    Message:= CONCAT('Expected stState.nBufferPos to equal ', TO_STRING(nExpectedBufferPos)));
    
AssertEquals_UDINT(
    Expected:= nExpectedFieldIndex,
    Actual:= fbRepeatedField.nCount,
    Message:= CONCAT('Expected fbRepeatedField.nCount to equal ', TO_STRING(nExpectedFieldIndex)));
END_METHOD

METHOD PRIVATE ShouldReadRepeatedFieldTheory : REFERENCE TO FB_Test
(*
    syntax = "proto3";
    
    message exampleMessage
    {
      repeated fixed32 repeatedFixed32 = 4;
    }
*)
VAR CONSTANT
    cRawValueZeroLength     : ARRAY[0..31] OF BYTE := [16#22, 16#00];       // field #4
    cRawValue1              : ARRAY[0..31] OF BYTE := [16#00, 16#22, 16#18, 16#00, 16#00, 16#00, 16#00, 16#D2, 16#04, 16#00, 16#00, 16#39, 16#05, 16#00, 16#00, 16#FF, 16#FF, 16#FF, 16#FF, 16#C7, 16#FA, 16#FF, 16#FF, 16#4E, 16#61, 16#BC, 16#00];
    
END_VAR

VAR CONSTANT
    aExpectedZeroLength     : ARRAY [0..7] OF DINT := [0, 0, 0, 0, 0, 0, 0, 0];
    aExpected1              : ARRAY [0..7] OF DINT := [0, 1234, 1337, -1, -1337, 12345678, 0, 0];
END_VAR
TEST(__POUNAME());

ShouldReadRepeatedField(aBuffer:= cRawValueZeroLength, aExpected:= aExpectedZeroLength, nBufferPosStart:= 0, nExpectedBufferPos:= 2, nExpectedFieldIndex:= 0, ipFieldCodec:= THIS^.fbFieldCodec);
ShouldReadRepeatedField(aBuffer:= cRawValue1, aExpected:= aExpected1, nBufferPosStart:= 1, nExpectedBufferPos:= 27, nExpectedFieldIndex:= 6, ipFieldCodec:= THIS^.fbFieldCodec);

TEST_FINISHED_NAMED(__POUNAME());
END_METHOD

END_FUNCTION_BLOCK

// ---- FieldCodec/FB_FieldCodecFixed32.TcPOU
FUNCTION_BLOCK FB_FieldCodecFixed32 EXTENDS FB_FieldCodec
VAR_INPUT
END_VAR
VAR_OUTPUT
END_VAR
VAR
    nValue : UDINT;
END_VAR

METHOD CalculatePackedDataSize : HRESULT
VAR_INPUT CONSTANT
	anyFirstElem	: T_Any;
	nLength	        : UDINT;        // items to write
END_VAR
VAR_OUTPUT
    nPackedDataSize : UDINT;
END_VAR
VAR
    anyItem         : T_ANY;
    i               : UDINT;
    nValue          : DINT;
END_VAR
anyItem := anyFirstElem;

IF nLength < 1 THEN
    nPackedDataSize := 0;
    RETURN;
END_IF

FOR i := 0  TO nLength - 1 DO
    anyItem.pValue := anyFirstElem.pValue + (i * TO_UDINT(anyFirstElem.diSize)); 
    nValue := PDINT_TO_DINT(anyItem.pValue);
    nPackedDataSize := nPackedDataSize + F_ComputeFixed32Size(TO_UDINT(nValue));
END_FOR
END_METHOD

METHOD IsPackedRepeatedField : BOOL
VAR_INPUT
	nTag	: UDINT;
END_VAR
IsPackedRepeatedField := F_IsPackedRepeatedField(nTag);
END_METHOD


METHOD ValueReader : HRESULT
VAR_IN_OUT      
    stCtx : ST_ParseContext;
END_VAR
VAR_OUTPUT
	anyOut	: T_Any;
END_VAR

ValueReader := F_ParseRawLittleEndian32(stCtx, nValue=> nValue);
anyOut := F_ToAnyType(anyArg:= nValue);
END_METHOD

METHOD ValueWriter : HRESULT
VAR_IN_OUT
    stCtx  : ST_WriteContext;
END_VAR
VAR_INPUT
    anyIn : T_ANY;
END_VAR
VAR
    nValue  : DINT;
END_VAR

nValue := PDINT_TO_DINT(anyIn.pValue);
ValueWriter := F_WriteFixed32(stCtx, TO_UDINT(nValue));
END_METHOD

END_FUNCTION_BLOCK

// ---- __TESTs/RepeatedFieldTests/Read/FB_ReadRepeatedFieldFixed64Tests.TcPOU
FUNCTION_BLOCK INTERNAL FINAL FB_ReadRepeatedFieldFixed64Tests EXTENDS FB_TestSuite
VAR_INPUT
END_VAR
VAR_OUTPUT
END_VAR
VAR
	aActual             : ARRAY [0..7] OF LINT;
    fbFieldCodec 		: FB_FieldCodecFixed64(nTag:= 16#0A);
	fbRepeatedField		: FB_RepeatedField(anyArray:= F_ToAnyType(aActual), anyFirstElem:= F_ToAnyType(aActual[0]), ipFieldCodec:= fbFieldCodec);
END_VAR

ShouldReadRepeatedFieldTheory();

METHOD PRIVATE Reset
VAR_INPUT
END_VAR
fbRepeatedField.Initialize();
MEMSET(destAddr:= ADR(aActual), fillByte:= 16#0, n:= SIZEOF(aActual));
END_METHOD

METHOD PRIVATE ShouldReadRepeatedField
VAR_IN_OUT CONSTANT
    aBuffer     : ARRAY [*] OF BYTE;
    aExpected   : ARRAY [*] OF LINT;
END_VAR
VAR_INPUT CONSTANT
    nBufferPosStart     : UDINT;
    nExpectedBufferPos  : UDINT;
    nExpectedFieldIndex : UDINT;
    ipFieldCodec        : I_FieldCodec;
END_VAR
VAR_INST
    fbCtx               : FB_ParseContext;
END_VAR
VAR
    hr                  : HRESULT;
    nTag                : UDINT;
END_VAR
// Arrange
Reset();
fbCtx.FromBuffer(aBuffer);
fbCtx.refCtx.stState.nBufferPos := nBufferPosStart;

// Act
F_ParseTag(fbCtx.refCtx, nTag=> nTag);
hr := fbRepeatedField.AddEntriesFrom(fbParseCtx:= fbCtx, ipFieldCodec:= ipFieldCodec);

// Assert
AssertEquals_DINT(
    Expected:= S_OK,
    Actual:= hr,
    Message:= 'Expected S_OK instead of error');
    
{warning disable C0041}
AssertArrayEquals_LINT(Expecteds:= aExpected, Actuals:= aActual, Message:= '');
 
AssertEquals_UDINT(
    Expected:= nExpectedBufferPos,
    Actual:= fbCtx.refCtx.stState.nBufferPos,
    Message:= CONCAT('Expected stState.nBufferPos to equal ', TO_STRING(nExpectedBufferPos)));
    
AssertEquals_UDINT(
    Expected:= nExpectedFieldIndex,
    Actual:= fbRepeatedField.nCount,
    Message:= CONCAT('Expected fbRepeatedField.nCount to equal ', TO_STRING(nExpectedFieldIndex)));
END_METHOD

METHOD PRIVATE ShouldReadRepeatedFieldTheory : REFERENCE TO FB_Test
(*
    syntax = "proto3";
    
    message exampleMessage
    {
      repeated fixed32 repeatedFixed32 = 4;
    }
*)
VAR CONSTANT
    cRawValueZeroLength     : ARRAY[0..31] OF BYTE := [16#22, 16#00];       // field #4
    cRawValue1              : ARRAY[0..100] OF BYTE := [16#22, 16#30, 16#00, 16#00, 16#00, 16#00, 16#00, 16#00, 16#00, 16#00, 16#d2, 16#04, 16#00, 16#00, 16#00, 16#00, 16#00, 16#00, 16#39, 16#05, 16#00, 16#00, 16#00, 16#00, 16#00, 16#00, 16#ff, 16#ff, 16#ff, 16#ff, 16#ff, 16#ff, 16#ff, 16#ff, 16#c7, 16#fa, 16#ff, 16#ff, 16#ff, 16#ff, 16#ff, 16#ff, 16#4e, 16#61, 16#bc, 16#00, 16#00, 16#00, 16#00, 16#00];
    
END_VAR

VAR CONSTANT
    aExpectedZeroLength     : ARRAY [0..7] OF LINT := [0, 0, 0, 0, 0, 0, 0, 0];
    aExpected1              : ARRAY [0..7] OF LINT := [0, 1234, 1337, -1, -1337, 12345678, 0, 0];
END_VAR
TEST(__POUNAME());

ShouldReadRepeatedField(aBuffer:= cRawValueZeroLength, aExpected:= aExpectedZeroLength, nBufferPosStart:= 0, nExpectedBufferPos:= 2, nExpectedFieldIndex:= 0, ipFieldCodec:= THIS^.fbFieldCodec);
ShouldReadRepeatedField(aBuffer:= cRawValue1, aExpected:= aExpected1, nBufferPosStart:= 0, nExpectedBufferPos:= 50, nExpectedFieldIndex:= 6, ipFieldCodec:= THIS^.fbFieldCodec);

TEST_FINISHED_NAMED(__POUNAME());
END_METHOD

END_FUNCTION_BLOCK

// ---- FieldCodec/FB_FieldCodecFixed64.TcPOU
FUNCTION_BLOCK FB_FieldCodecFixed64 EXTENDS FB_FieldCodec
VAR_INPUT
END_VAR
VAR_OUTPUT
END_VAR
VAR
    nValue : ULINT;
END_VAR

METHOD CalculatePackedDataSize : HRESULT
VAR_INPUT CONSTANT
	anyFirstElem	: T_Any;
	nLength	        : UDINT;        // items to write
END_VAR
VAR_OUTPUT
    nPackedDataSize : UDINT;
END_VAR
VAR
    anyItem         : T_ANY;
    i               : UDINT;
    nValue          : LINT;
END_VAR
anyItem := anyFirstElem;

IF nLength < 1 THEN
    nPackedDataSize := 0;
    RETURN;
END_IF

FOR i := 0  TO nLength - 1 DO
    anyItem.pValue := anyFirstElem.pValue + (i * TO_UDINT(anyFirstElem.diSize)); 
    nValue := PLINT_TO_LINT(anyItem.pValue);
    nPackedDataSize := nPackedDataSize + F_ComputeFixed64Size(TO_ULINT(nValue));
END_FOR
END_METHOD

METHOD IsPackedRepeatedField : BOOL
VAR_INPUT
	nTag	: UDINT;
END_VAR
IsPackedRepeatedField := F_IsPackedRepeatedField(nTag);
END_METHOD


METHOD ValueReader : HRESULT
VAR_IN_OUT      
    stCtx : ST_ParseContext;
END_VAR
VAR_OUTPUT
	anyOut	: T_Any;
END_VAR

ValueReader := F_ParseRawLittleEndian64(stCtx, nValue=> nValue);
anyOut := F_ToAnyType(anyArg:= nValue);
END_METHOD

METHOD ValueWriter : HRESULT
VAR_IN_OUT
    stCtx  : ST_WriteContext;
END_VAR
VAR_INPUT
    anyIn : T_ANY;
END_VAR
VAR
    nValue  : LINT;
END_VAR

nValue := PLINT_TO_LINT(anyIn.pValue);
ValueWriter := F_WriteFixed64(stCtx, TO_ULINT(nValue));
END_METHOD

END_FUNCTION_BLOCK

// ---- __TESTs/RepeatedFieldTests/Read/FB_ReadRepeatedFieldStringTests.TcPOU
FUNCTION_BLOCK INTERNAL FINAL FB_ReadRepeatedFieldStringTests EXTENDS FB_TestSuite
VAR_INPUT
END_VAR
VAR_OUTPUT
END_VAR
VAR
	aActual             : ARRAY[0..15] OF T_MAXSTRING;
	fbFieldCodec 		: FB_FieldCodecString(nTag:= 16#0A);
	fbRepeatedField		: FB_RepeatedField(anyArray:= F_ToAnyType(aActual), anyFirstElem:= F_ToAnyType(aActual[0]), ipFieldCodec:= fbFieldCodec);
END_VAR

ShouldReadRepeatedFieldTheory();

METHOD PRIVATE Reset
VAR_INPUT
END_VAR
fbRepeatedField.Initialize();
MEMSET(destAddr:= ADR(aActual), fillByte:= 16#0, n:= SIZEOF(aActual));
END_METHOD

METHOD PRIVATE ShouldReadRepeatedField
VAR_IN_OUT CONSTANT
    aBuffer     : ARRAY [*] OF BYTE;
    aExpected   : ARRAY [*] OF T_MAXSTRING;
END_VAR
VAR_INPUT CONSTANT
    nBufferPosStart     : UDINT;
    nExpectedBufferPos  : UDINT;
    nExpectedFieldIndex : UDINT;
    ipFieldCodec        : I_FieldCodec;
END_VAR
VAR_INST
    fbCtx               : FB_ParseContext;
END_VAR
VAR
    
    hr                  : HRESULT;
    nTag                : UDINT;
    i                   : DINT;
    aTmpBuffer          : ARRAY[0..1023] OF BYTE := [SIZEOF(aTmpBuffer)(16#FF)];
END_VAR
// Arrange
Reset();
fbCtx.FromBuffer(aBuffer);
fbCtx.refCtx.stState.nBufferPos := nBufferPosStart;

THIS^.fbFieldCodec.SetTmpBuffer(anyString:= F_ToAnyBytes(aTmpBuffer));

// Act
F_ParseTag(fbCtx.refCtx, nTag=> nTag);
hr := fbRepeatedField.AddEntriesFrom(fbParseCtx:= fbCtx, ipFieldCodec:= ipFieldCodec);

// Assert
AssertEquals_DINT(
    Expected:= S_OK,
    Actual:= hr,
    Message:= 'Expected S_OK instead of error');
    
{warning disable C0041}
// AssertArrayEquals_(Expecteds:= aExpected, Actuals:= aActual, Message:= '');
FOR i := 0  TO UPPER_BOUND(aExpected, 1) DO 
    AssertEquals_STRING(Expected:= aExpected[i], Actual:= aActual[i], Message:= '');
END_FOR

AssertEquals_UDINT(
    Expected:= nExpectedBufferPos,
    Actual:= fbCtx.refCtx.stState.nBufferPos,
    Message:= CONCAT('Expected stState.nBufferPos to equal ', TO_STRING(nExpectedBufferPos)));
    
AssertEquals_UDINT(
    Expected:= nExpectedFieldIndex,
    Actual:= fbRepeatedField.nCount,
    Message:= CONCAT('Expected fbRepeatedField.nCount to equal ', TO_STRING(nExpectedFieldIndex)));
END_METHOD

METHOD PRIVATE ShouldReadRepeatedFieldTheory : REFERENCE TO FB_Test
VAR CONSTANT
    cRawValueString1    : ARRAY[0..255] OF BYTE := [16#0A, 16#0B, 16#54, 16#65, 16#73, 16#74, 16#53, 16#74, 16#72, 16#69, 16#6E, 16#67, 16#30, 16#0A, 16#0B, 16#54, 16#65, 16#73, 16#74, 16#53, 16#74, 16#72, 16#69, 16#6E, 16#67, 16#31, 16#0A, 16#0B, 16#54, 16#65, 16#73, 16#74, 16#53, 16#74, 16#72, 16#69, 16#6E, 16#67, 16#32, 16#0A, 16#0B, 16#54, 16#65, 16#73, 16#74, 16#53, 16#74, 16#72, 16#69, 16#6E, 16#67, 16#33];
    
END_VAR

VAR CONSTANT
    aExpectedString1        : ARRAY[0..15] OF T_MAXSTRING := ['TestString0', 'TestString1', 'TestString2', 'TestString3'];
END_VAR
TEST(__POUNAME());

ShouldReadRepeatedField(aBuffer:= cRawValueString1, aExpected:= aExpectedString1, nBufferPosStart:= 0, nExpectedBufferPos:= 53, nExpectedFieldIndex:= 4, THIS^.fbFieldCodec);

TEST_FINISHED_NAMED(__POUNAME());
END_METHOD

END_FUNCTION_BLOCK

// ---- FieldCodec/FB_FieldCodecString.TcPOU
FUNCTION_BLOCK FB_FieldCodecString EXTENDS FB_FieldCodec
VAR_INPUT
END_VAR
VAR_OUTPUT
END_VAR
VAR
    sValue      	: T_MAXSTRING;
    anyStringTmp : T_AnyString;
END_VAR

{attribute 'analysis' := '-33'}
METHOD CalculatePackedDataSize : HRESULT
VAR_INPUT CONSTANT
	anyFirstElem	: T_Any;
	nLength	        : UDINT;        // items to write
END_VAR
VAR_OUTPUT
    nPackedDataSize : UDINT;
END_VAR

CalculatePackedDataSize := 0;
END_METHOD

METHOD IsPackedRepeatedField : BOOL
VAR_INPUT
    {attribute 'analysis' := '-33' } 
	nTag	: UDINT;
END_VAR

IsPackedRepeatedField := FALSE;
END_METHOD

// Needs to be called, if destination string is larger then T_MAXSTRING.
METHOD INTERNAL SetTmpBuffer
VAR_INPUT
    anyString : T_AnyString;
END_VAR
anyStringTmp := anyString;
END_METHOD


METHOD ValueReader : HRESULT
VAR_IN_OUT
    stCtx : ST_ParseContext;
END_VAR
VAR_OUTPUT
	anyOut	: T_Any;
END_VAR
IF anyStringTmp.pValue <> NULL THEN
    anyOut := anyStringTmp;
ELSE
    anyOut := F_ToAnyString(sValue);
END_IF
ValueReader := F_ReadString(stCtx, anyOut);
END_METHOD

METHOD ValueWriter : HRESULT
VAR_IN_OUT
    stCtx  : ST_WriteContext;
END_VAR
VAR_INPUT
    anyIn : T_ANY;
END_VAR

ValueWriter := F_WriteRawString(stCtx, anyIn);
END_METHOD

END_FUNCTION_BLOCK

// ---- Helper/POUs/F_ToAnyString.TcPOU
FUNCTION F_ToAnyString : T_AnyString
VAR_INPUT
    anyArg	: ANY_STRING;
END_VAR

F_ToAnyString := anyArg;

END_FUNCTION

// ---- __TESTs/RepeatedFieldTests/Write/PRG_WriteRepeatedFieldTests.TcPOU
{attribute 'analysis' := '-33'}
PROGRAM INTERNAL PRG_WriteRepeatedFieldTests
{IF defined (UNIT_TEST)}
	fbWriteRepeatedFieldBoolTests : FB_WriteRepeatedFieldBoolTests;
	fbWriteRepeatedFieldBytesTests : FB_WriteRepeatedFieldBytesTests;
//     fbWriteRepeatedFieldDoubleTests : FB_WriteRepeatedFieldDoubleTests;
// 	fbWriteRepeatedFieldFixed32Tests : FB_WriteRepeatedFieldFixed32Tests;
//     fbWriteRepeatedFieldFixed64Tests : FB_WriteRepeatedFieldFixed64Tests;
// 	fbWriteRepeatedFieldFloatTests : FB_WriteRepeatedFieldFloatTests;
//     fbWriteRepeatedFieldInt32Tests : FB_WriteRepeatedFieldInt32Tests;
//     fbWriteRepeatedFieldInt64Tests : FB_WriteRepeatedFieldInt64Tests;
//     fbWriteRepeatedFieldSInt32Tests : FB_WriteRepeatedFieldSInt32Tests;
//     fbWriteRepeatedFieldSInt64Tests : FB_WriteRepeatedFieldSInt64Tests;
//     fbWriteRepeatedFieldStringTests : FB_WriteRepeatedFieldStringTests;
// 	fbWriteRepeatedFieldUint32Tests : FB_WriteRepeatedFieldUint32Tests;
// 	fbWriteRepeatedFieldUint64Tests : FB_WriteRepeatedFieldUint64Tests;
// 	fbWriteRepeatedFieldMessageTests : FB_WriteRepeatedFieldMessageTests;
{END_IF}

END_PROGRAM

// ---- __TESTs/RepeatedFieldTests/Write/FB_WriteRepeatedFieldBoolTests.TcPOU
FUNCTION_BLOCK INTERNAL FINAL FB_WriteRepeatedFieldBoolTests EXTENDS FB_TestSuite
VAR_INPUT
END_VAR
VAR_OUTPUT
END_VAR
VAR
	aActual             : ARRAY [0..15] OF BOOL;
    fbFieldCodec 		: FB_FieldCodecBool(nTag:= 16#0A);
	fbRepeatedField		: FB_RepeatedField(anyArray:= F_ToAnyType(aActual), anyFirstElem:= F_ToAnyType(aActual[0]), ipFieldCodec:= fbFieldCodec);
END_VAR

ShouldWriteRepeatedFieldTheory();

METHOD PRIVATE Reset
VAR_INPUT
END_VAR
fbRepeatedField.Initialize();
MEMSET(destAddr:= ADR(aActual), fillByte:= 16#0, n:= SIZEOF(aActual));
END_METHOD

METHOD PRIVATE ShouldWriteRepeatedField
VAR_IN_OUT CONSTANT
    aExpected   : ARRAY [*] OF BYTE;
END_VAR
VAR_INPUT
	aValues     : ARRAY [0..15] OF BOOL;
    nLength     : UDINT;
    nTag        : UDINT;
    nBufferPosStart     : UDINT;
    nExpectedBufferPos  : UDINT;
    ipFieldCodec        : I_FieldCodec;
END_VAR
VAR_INST
    fbCtx   : FB_WriteContext;
END_VAR
VAR
    aActualBuffer       : ARRAY [0..15] OF BYTE;
    hr                  : HRESULT;
END_VAR
// Arrange
Reset();
fbCtx.FromBuffer(aActualBuffer);
fbCtx.refCtx.stState.nBufferPos := nBufferPosStart;
fbRepeatedField.InitializeFromArray(anyArray:= F_ToAnyType(aValues), anyFirstElem:= F_ToAnyType(aValues[0]), nCount:= nLength);
// Act
hr := fbRepeatedField.WriteTo(fbWriteCtx:= fbCtx, ipFieldCodec:= ipFieldCodec);

// Assert
AssertEquals_DINT(
    Expected:= S_OK,
    Actual:= hr,
    Message:= 'Expected S_OK instead of error');
    
{warning disable C0041}
AssertArrayEquals_BYTE(Expecteds:= aExpected, Actuals:= aActualBuffer, Message:= '');
 
AssertEquals_UDINT(
    Expected:= nExpectedBufferPos,
    Actual:= fbCtx.refCtx.stState.nBufferPos,
    Message:= CONCAT('Expected stState.nBufferPos to equal ', TO_STRING(nExpectedBufferPos)));
END_METHOD

METHOD PRIVATE ShouldWriteRepeatedFieldTheory : REFERENCE TO FB_Test
VAR CONSTANT
    cExpectedZeroLength		: ARRAY[0..15] OF BYTE := [16#00, 16#00];
    cExpected1        		: ARRAY[0..15] OF BYTE := [16#00, 16#0A, 16#05, 16#01, 16#00, 16#01, 16#01, 16#00];
END_VAR

VAR CONSTANT
    aZeroLength    			: ARRAY [0..15] OF BOOL := [0, 0, 0, 0, 0, 0, 0, 0, 0, 0, 0, 0, 0, 0, 0, 0];
    aValue1              	: ARRAY [0..15] OF BOOL := [TRUE, FALSE, TRUE, TRUE, FALSE];
END_VAR
TEST(__POUNAME());

ShouldWriteRepeatedField(aExpected:= cExpectedZeroLength, aValues:= aZeroLength, nLength:= 0, nTag:= 1, nBufferPosStart:= 0, nExpectedBufferPos:= 0, ipFieldCodec:= THIS^.fbFieldCodec);
ShouldWriteRepeatedField(aExpected:= cExpected1, aValues:= aValue1, nLength:= 5, nTag:= 1, nBufferPosStart:= 1, nExpectedBufferPos:= 8, ipFieldCodec:= THIS^.fbFieldCodec);

TEST_FINISHED_NAMED(__POUNAME());
END_METHOD

END_FUNCTION_BLOCK

// ---- __TESTs/RepeatedFieldTests/Write/FB_WriteRepeatedFieldBytesTests.TcPOU
FUNCTION_BLOCK INTERNAL FINAL FB_WriteRepeatedFieldBytesTests EXTENDS FB_TestSuite
VAR_INPUT
END_VAR
VAR_OUTPUT
END_VAR
VAR
	aActual             : ARRAY[0..3] OF ARRAY[0..4] OF BYTE;
    fbFieldCodec 		: FB_FieldCodecBytes(nTag:= 16#0A);
	fbRepeatedField		: FB_RepeatedField(anyArray:= F_ToAnyType(aActual), anyFirstElem:= F_ToAnyType(aActual[0]), ipFieldCodec:= fbFieldCodec);
END_VAR

ShouldWriteRepeatedFieldTheory();

METHOD PRIVATE Reset
VAR_INPUT
END_VAR
fbRepeatedField.Initialize();
MEMSET(destAddr:= ADR(aActual), fillByte:= 16#0, n:= SIZEOF(aActual));
END_METHOD

METHOD PRIVATE ShouldWriteRepeatedField
VAR_IN_OUT CONSTANT
    aExpected   : ARRAY [*] OF BYTE;
END_VAR
VAR_INPUT
    aValues     : ARRAY[0..3] OF ARRAY[0..4] OF BYTE;
    nLength     : UDINT;
    nTag 		: UDINT;
    nBufferPosStart     : UDINT;
    nExpectedBufferPos  : UDINT;
    ipFieldCodec        : I_FieldCodec;
END_VAR
VAR_INST
    fbCtx   : FB_WriteContext;
END_VAR
VAR
    aActualBuffer       : ARRAY [0..63] OF BYTE;
    hr                  : HRESULT;
END_VAR
// Arrange
Reset();
fbCtx.FromBuffer(aActualBuffer);
fbCtx.refCtx.stState.nBufferPos := nBufferPosStart;
ipFieldCodec.Tag := nTag;
fbRepeatedField.InitializeFromArray(anyArray:= F_ToAnyType(aValues), anyFirstElem:= F_ToAnyType(aValues[0]), nCount:= nLength);

// Act
hr := fbRepeatedField.WriteTo(fbWriteCtx:= fbCtx, ipFieldCodec:= ipFieldCodec);

// Assert
AssertEquals_DINT(
    Expected:= S_OK,
    Actual:= hr,
    Message:= 'Expected S_OK instead of error');
    
{warning disable C0041}
AssertArrayEquals_BYTE(Expecteds:= aExpected, Actuals:= aActualBuffer, Message:= '');
 
AssertEquals_UDINT(
    Expected:= nExpectedBufferPos,
    Actual:= fbCtx.refCtx.stState.nBufferPos,
    Message:= CONCAT('Expected stState.nBufferPos to equal ', TO_STRING(nExpectedBufferPos)));
END_METHOD

METHOD PRIVATE ShouldWriteRepeatedFieldTheory : REFERENCE TO FB_Test
VAR CONSTANT
    aExpectedBufferZeroLen  : ARRAY[0..63] OF BYTE := [16#00, 16#00];
    aExpectedBuffer1        : ARRAY[0..63] OF BYTE := [16#00, 16#1A, 16#05, 16#00, 16#FF, 16#01, 16#00, 16#00, 16#1A, 16#05, 16#2A, 16#45, 16#7B, 16#00, 16#FF];
END_VAR

VAR CONSTANT
    aValueZeroLen           : ARRAY[0..3] OF ARRAY[0..4] OF BYTE := [];
    aValue1                 : ARRAY[0..3] OF ARRAY[0..4] OF BYTE := [[0, 255, 1], [42, 69, 123, 0 , 255]];
END_VAR
TEST(__POUNAME());
ShouldWriteRepeatedField(aExpected:= aExpectedBufferZeroLen, aValues:= aValueZeroLen, nLength:= 0, nTag:= F_MakeTag(1, E_WireType.LengthDelimited), nBufferPosStart:= 0, nExpectedBufferPos:= 0, ipFieldCodec:= THIS^.fbFieldCodec);
ShouldWriteRepeatedField(aExpected:= aExpectedBuffer1, aValues:= aValue1, nLength:= 2, nTag:= F_MakeTag(3, E_WireType.LengthDelimited), nBufferPosStart:= 1, nExpectedBufferPos:= 15, ipFieldCodec:= THIS^.fbFieldCodec);
TEST_FINISHED_NAMED(__POUNAME());
END_METHOD

END_FUNCTION_BLOCK

// ---- __TESTs/RepeatedFieldTests/RoundTrip/PRG_RoundTripRepeatedFieldTests.TcPOU
{attribute 'analysis' := '-33'}
PROGRAM INTERNAL PRG_RoundTripRepeatedFieldTests
VAR
{IF defined (UNIT_TEST)}
	fbRoundTripRepeatedFieldUInt32Tests		: FB_RoundTripRepeatedFieldUInt32Tests;
	fbRoundTripRepeatedFieldUInt64Tests		: FB_RoundTripRepeatedFieldUInt64Tests;
	fbRoundTripRepeatedFieldStringTests		: FB_RoundTripRepeatedFieldStringTests;
{END_IF}
END_VAR

END_PROGRAM

// ---- __TESTs/RepeatedFieldTests/RoundTrip/FB_RoundTripRepeatedFieldUInt32Tests.TcPOU
FUNCTION_BLOCK INTERNAL FINAL FB_RoundTripRepeatedFieldUInt32Tests EXTENDS FB_TestSuite
VAR CONSTANT
    cExpected 			: ARRAY[0..7] OF UDINT := [0, 42, 6969, 1337, 123456789];
	cExpectedFieldIndex : UDINT := 5;
END_VAR
VAR
    aBuffer         	: ARRAY[0..255] OF BYTE;
    hrWriterActual  	: HRESULT;
    hrParserActual  	: HRESULT;
	aActuals,aValues	: ARRAY[0..7] OF UDINT ;
	nActualTag			: UDINT;
	nExpectedTag	    : UDINT;
	fbParseCtx_SUT      : FB_ParseContext;
	fbWriteCtx_SUT  	: FB_WriteContext;
	fbFieldCodec 		: FB_FieldCodecUint32(nTag:= F_MakeTag(nFieldNumber:= 3, eWireType:= E_WireType.LengthDelimited));
	fbRepeatedField_Write : FB_RepeatedField(anyArray := F_ToAnyType(aValues), anyFirstElem:= F_ToAnyType(aValues[0]), ipFieldCodec:= fbFieldCodec);
	fbRepeatedField_Parse : FB_RepeatedField(anyArray:= F_ToAnyType(aActuals), anyFirstElem:= F_ToAnyType(aActuals[0]), ipFieldCodec:= fbFieldCodec);	
END_VAR

TEST(__POUNAME());

// Arrange
nExpectedTag := F_MakeTag(nFieldNumber:= 3, eWireType:= E_WireType.LengthDelimited);
aValues := cExpected;
fbRepeatedField_Write.InitializeFromArray(anyArray:= F_ToAnyType(aValues), anyFirstElem:= F_ToAnyType(aValues[0]), nCount:= 5);

fbWriteCtx_SUT.FromBuffer(aBuffer);
fbParseCtx_SUT.FromBuffer(aBuffer);

// Act

hrWriterActual := fbRepeatedField_Write.WriteTo(fbWriteCtx_SUT, fbFieldCodec);
fbParseCtx_SUT.ReadTag(nTag=> nActualTag);
hrParserActual := fbRepeatedField_Parse.AddEntriesFrom(fbParseCtx_SUT, fbFieldCodec);

// Assert

AssertEquals_DINT(Expected:= S_OK, Actual:= hrWriterActual, Message:= 'Expected hrWriterActual = S_OK');
AssertEquals_DINT(Expected:= S_OK, Actual:= hrParserActual, Message:= 'Expected hrParserActual = S_OK');
AssertEquals_UDINT(Expected:= nExpectedTag, Actual:= nActualTag, Message:= 'Expeced nActualTag to equal nExpectedTag.');
AssertEquals_UDINT(Expected:= cExpectedFieldIndex, Actual:= fbRepeatedField_Parse.nCount, Message:= 'Expeced fbRepeatedField_Parse.nCount to equal cExpectedFieldIndex.');
{warning disable C0041}
AssertArrayEquals_UDINT(Expecteds:= cExpected, Actuals:= aActuals, Message:= '');

TEST_FINISHED_NAMED(__POUNAME());

END_FUNCTION_BLOCK

// ---- __TESTs/RepeatedFieldTests/RoundTrip/FB_RoundTripRepeatedFieldUInt64Tests.TcPOU
FUNCTION_BLOCK INTERNAL FINAL FB_RoundTripRepeatedFieldUInt64Tests EXTENDS FB_TestSuite
VAR CONSTANT
    cExpected 			: ARRAY[0..7] OF ULINT := [0, 42, 6969, 1337, 16#FFFFFFFFFFFFFFFF];
	cExpectedFieldIndex : UDINT := 5;
END_VAR
VAR
    aBuffer         	: ARRAY[0..255] OF BYTE;
    hrWriterActual  	: HRESULT;
    hrParserActual  	: HRESULT;
	aActuals,aValues	: ARRAY[0..7] OF ULINT ;
	nActualTag			: UDINT;
	nExpectedTag	    : UDINT;
	fbParseCtx_SUT      : FB_ParseContext;
	fbWriteCtx_SUT      : FB_WriteContext;
	fbFieldCodec 		: FB_FieldCodecUint64(nTag:= F_MakeTag(nFieldNumber:= 3, eWireType:= E_WireType.LengthDelimited));
	fbRepeatedField_Write : FB_RepeatedField(anyArray:= F_ToAnyType(aValues), anyFirstElem:= F_ToAnyType(aValues[0]), ipFieldCodec:= fbFieldCodec);
	fbRepeatedField_Parse : FB_RepeatedField(anyArray:= F_ToAnyType(aActuals), anyFirstElem:= F_ToAnyType(aActuals[0]), ipFieldCodec:= fbFieldCodec);	
END_VAR

TEST(__POUNAME());

// Arrange
nExpectedTag := F_MakeTag(nFieldNumber:= 3, eWireType:= E_WireType.LengthDelimited);
aValues := cExpected;
fbRepeatedField_Write.InitializeFromArray(anyArray:= F_ToAnyType(aValues), anyFirstElem:= F_ToAnyType(aValues[0]), nCount:= 5);
fbWriteCtx_SUT.FromBuffer(aBuffer);
fbParseCtx_SUT.FromBuffer(aBuffer);

// Act

hrWriterActual := fbRepeatedField_Write.WriteTo(fbWriteCtx_SUT, fbFieldCodec);
fbParseCtx_SUT.ReadTag(nTag=> nActualTag);
hrParserActual := fbRepeatedField_Parse.AddEntriesFrom(fbParseCtx_SUT, fbFieldCodec);

// Assert

AssertEquals_DINT(Expected:= S_OK, Actual:= hrWriterActual, Message:= 'Expected hrWriterActual = S_OK');
AssertEquals_DINT(Expected:= S_OK, Actual:= hrParserActual, Message:= 'Expected hrParserActual = S_OK');
AssertEquals_UDINT(Expected:= nExpectedTag, Actual:= nActualTag, Message:= 'Expeced nActualTag to equal nExpectedTag.');
AssertEquals_UDINT(Expected:= cExpectedFieldIndex, Actual:= fbRepeatedField_Parse.nCount, Message:= 'Expeced fbRepeatedField_Parse.nCount to equal cExpectedFieldIndex.');
{warning disable C0041}
AssertArrayEquals_ULINT(Expecteds:= cExpected, Actuals:= aActuals, Message:= '');

TEST_FINISHED_NAMED(__POUNAME());

END_FUNCTION_BLOCK

// ---- FieldCodec/FB_FieldCodecUInt64.TcPOU
FUNCTION_BLOCK FB_FieldCodecUInt64 EXTENDS FB_FieldCodec
VAR_INPUT
END_VAR
VAR_OUTPUT
END_VAR
VAR
    nValue : ULINT;
END_VAR

METHOD CalculatePackedDataSize : HRESULT
VAR_INPUT CONSTANT
	anyFirstElem	: T_Any;
	nLength	        : UDINT;        // items to write
END_VAR
VAR_OUTPUT
    nPackedDataSize : UDINT;
END_VAR
VAR
    anyItem         : T_ANY;
    i               : UDINT;
    nValue          : ULINT;
END_VAR
anyItem := anyFirstElem;

IF nLength < 1 THEN
    nPackedDataSize := 0;
    RETURN;
END_IF

FOR i := 0  TO nLength - 1 DO
    anyItem.pValue := anyFirstElem.pValue + (i * TO_UDINT(anyFirstElem.diSize)); 
    MEMCPY(destAddr:= ADR(nValue), srcAddr:= anyItem.pValue, n:= TO_UDINT(anyFirstElem.diSize));
    nPackedDataSize := nPackedDataSize + F_ComputeUInt64Size(nValue);
END_FOR
END_METHOD

METHOD IsPackedRepeatedField : BOOL
VAR_INPUT
	nTag	: UDINT;
END_VAR
IsPackedRepeatedField := F_IsPackedRepeatedField(nTag);
END_METHOD


METHOD ValueReader : HRESULT
VAR_IN_OUT      
    stCtx : ST_ParseContext;
END_VAR
VAR_OUTPUT
	anyOut	: T_Any;
END_VAR

ValueReader := F_ParseRawVarint64(stCtx, nValue);
anyOut := F_ToAnyType(anyArg:= nValue);
END_METHOD

METHOD ValueWriter : HRESULT
VAR_IN_OUT
    stCtx  : ST_WriteContext;
END_VAR
VAR_INPUT
    anyIn : T_ANY;
END_VAR
VAR
    nValue  : ULINT;
END_VAR

// nValue := PULINT_TO_ULINT(anyIn.pValue);
MEMCPY(destAddr:= ADR(nValue), srcAddr:= anyIn.pValue, n:= TO_UDINT(anyIn.diSize));
ValueWriter := F_WriteUInt64(stCtx, nValue);
END_METHOD

END_FUNCTION_BLOCK

// ---- __TESTs/RepeatedFieldTests/RoundTrip/FB_RoundTripRepeatedFieldStringTests.TcPOU
FUNCTION_BLOCK INTERNAL FINAL FB_RoundTripRepeatedFieldStringTests EXTENDS FB_TestSuite
VAR CONSTANT
    cExpected 			: ARRAY[0..7] OF STRING := ['abc', '123', '🤖👾�', 'ABCDEFG HIJK', 'äöüß'];
	cExpectedFieldIndex : UDINT := 5;
END_VAR
VAR
    aBuffer         	: ARRAY[0..255] OF BYTE;
    hrWriterActual  	: HRESULT;
    hrParserActual  	: HRESULT;
	aActuals, aValues	: ARRAY[0..7] OF STRING ;
	nActualTag			: UDINT;
	nExpectedTag	    : UDINT;
    fbParseCtx_SUT      : FB_ParseContext;
	fbWriteCtx_SUT		: FB_WriteContext;
	fbFieldCodec 		: FB_FieldCodecString(nTag:= F_MakeTag(nFieldNumber:= 3, eWireType:= E_WireType.LengthDelimited));
	fbRepeatedField_Write : FB_RepeatedField(anyArray:= F_ToAnyType(aValues), anyFirstElem:= F_ToAnyType(aValues[0]), ipFieldCodec:= fbFieldCodec);
	fbRepeatedField_Parse : FB_RepeatedField(anyArray:= F_ToAnyType(aActuals), anyFirstElem:= F_ToAnyType(aActuals[0]), ipFieldCodec:= fbFieldCodec);
END_VAR
VAR_TEMP
	i : INT;
END_VAR

TEST(__POUNAME());

// Arrange
nExpectedTag := F_MakeTag(nFieldNumber:= 3, eWireType:= E_WireType.LengthDelimited);
aValues := cExpected;
fbRepeatedField_Write.InitializeFromArray(anyArray:= F_ToAnyType(aValues), anyFirstElem:= F_ToAnyType(aValues[0]), nCount:= 5);
fbWriteCtx_SUT.FromBuffer(aBuffer);
fbParseCtx_SUT.FromBuffer(aBuffer);

// Act

hrWriterActual := fbRepeatedField_Write.WriteTo(fbWriteCtx_SUT, fbFieldCodec);
fbParseCtx_SUT.ReadTag(nTag=> nActualTag);
hrParserActual := fbRepeatedField_Parse.AddEntriesFrom(fbParseCtx_SUT, fbFieldCodec);

// Assert

AssertEquals_DINT(Expected:= S_OK, Actual:= hrWriterActual, Message:= 'Expected hrWriterActual = S_OK');
AssertEquals_DINT(Expected:= S_OK, Actual:= hrParserActual, Message:= 'Expected hrParserActual = S_OK');
AssertEquals_UDINT(Expected:= nExpectedTag, Actual:= nActualTag, Message:= 'Expeced nActualTag to equal nExpectedTag.');
AssertEquals_UDINT(Expected:= cExpectedFieldIndex, Actual:= fbRepeatedField_Parse.nCount, Message:= 'Expeced fbRepeatedField_Parse.nCount to equal cExpectedFieldIndex.');

FOR i := 0 TO 7 DO 
	AssertEquals_STRING(Expected:= cExpected[i], Actual:= aActuals[i], Message:= CONCAT(CONCAT('Index ', TO_STRING(i)), ' differ'));
END_FOR

TEST_FINISHED_NAMED(__POUNAME());

END_FUNCTION_BLOCK

// ---- __TESTs/HelperTests/PRG_HelperTests.TcPOU
{attribute 'analysis' := '-33'}
PROGRAM PRG_HelperTests
VAR
{IF defined (UNIT_TEST)}
    fbF_ToAnyBytesTests        : FB_F_ToAnyBytesTests;
{END_IF}
END_VAR

END_PROGRAM

// ---- __TESTs/HelperTests/FB_F_ToAnyBytesTests.TcPOU
FUNCTION_BLOCK INTERNAL FINAL FB_F_ToAnyBytesTests EXTENDS FB_TestSuite
VAR_INPUT
END_VAR
VAR_OUTPUT
END_VAR
VAR
END_VAR

ShouldConvertTheory();

METHOD PRIVATE ShouldConvert
VAR_IN_OUT CONSTANT
    aBytes : ARRAY [*] OF BYTE; 
END_VAR
VAR_INPUT
    anyBytesExpected : ANY;   
END_VAR

VAR
    
    anyBytesActual  : T_AnyBytes;
END_VAR

// Arrange

// Act

anyBytesActual := F_ToAnyBytes(aBytes);

// Assert

AssertEquals_DINT(
    Expected:= anyBytesExpected.diSize,
    Actual:= anyBytesActual.diSize,
    Message:= 'Sizes differ');
    
AssertTrue(
    Condition:= anyBytesExpected.TypeClass = anyBytesActual.TypeClass AND anyBytesExpected.TypeClass = __SYSTEM.TYPE_CLASS.TYPE_ARRAY,
    Message:= 'Expected TypeClass to equal TYPE_ARRAY');

AssertTrue(
    Condition:= anyBytesExpected.pValue = anyBytesActual.pValue,
    Message:= 'Pointer differ');
END_METHOD

METHOD PRIVATE ShouldConvertTheory
VAR_INPUT
END_VAR
VAR
    aBytes0 : ARRAY[0..0] OF BYTE := [];
    aBytes1 : ARRAY[0..42] OF BYTE := [];
    aBytes2 : ARRAY[-42..0] OF BYTE := [];
    aBytes3 : ARRAY[-42..42] OF BYTE := [];
    aBytes4 : ARRAY[-8..-1] OF BYTE := [];
END_VAR
TEST(__POUNAME());
ShouldConvert(aBytes:= aBytes0, anyBytesExpected:= aBytes0);
ShouldConvert(aBytes:= aBytes1, anyBytesExpected:= aBytes1);
ShouldConvert(aBytes:= aBytes2, anyBytesExpected:= aBytes2);
ShouldConvert(aBytes:= aBytes3, anyBytesExpected:= aBytes3);
ShouldConvert(aBytes:= aBytes4, anyBytesExpected:= aBytes4);
TEST_FINISHED_NAMED(__POUNAME());
END_METHOD

END_FUNCTION_BLOCK

// ---- __TESTs/SpanTests/PRG_SpanTests.TcPOU
{attribute 'analysis' := '-33'}
PROGRAM PRG_SpanTests
VAR
{IF defined (UNIT_TEST)}
    fbF_SpanFromArrayTests    : FB_F_SpanFromArrayTests;
    fbF_SpanSliceTests        : FB_F_SpanSliceTests;
{END_IF}
END_VAR

END_PROGRAM

// ---- __TESTs/SpanTests/FB_F_SpanFromArrayTests.TcPOU
FUNCTION_BLOCK FB_F_SpanFromArrayTests EXTENDS FB_TestSuite
VAR_INPUT
END_VAR
VAR_OUTPUT
END_VAR
VAR
    aBuffer1    : ARRAY[-3..3] OF BYTE;
    stActual    : ST_Span;
END_VAR

TEST(__POUNAME());

//Arrange

// Act
stActual := F_SpanFromArray(aBuffer:= aBuffer1);

//Assert
AssertEquals_ULINT(Expected:= ADR(aBuffer1), Actual:= stActual.pBuffer, Message:= '');
AssertEquals_UDINT(Expected:= 7, Actual:= stActual.nSize, Message:= '');

TEST_FINISHED_NAMED(__POUNAME());

END_FUNCTION_BLOCK

// ---- __TESTs/SpanTests/FB_F_SpanSliceTests.TcPOU
FUNCTION_BLOCK FB_F_SpanSliceTests EXTENDS FB_TestSuite
VAR_INPUT
END_VAR
VAR_OUTPUT
END_VAR
VAR
    stFromSpan  : ST_Span;
    stActual    : ST_Span;
END_VAR

TEST(__POUNAME());

stFromSpan.pBuffer := 123;
stFromSpan.nSize   := 32;

stActual := F_SpanSlice(stSpan:= stFromSpan, nStart:= 6, nLength:= 24);
AssertEquals_ULINT(Expected:= 129, Actual:= stActual.pBuffer, Message:= 'Valid Slice /w start 6');
AssertEquals_UDINT(Expected:= 24, Actual:= stActual.nSize, Message:= 'Valid Slice /w length 24');

stActual := F_SpanSlice(stSpan:= stFromSpan, nStart:= 0, nLength:= 32);
AssertEquals_ULINT(Expected:= 123, Actual:= stActual.pBuffer, Message:= 'Valid Slice /w start 0');
AssertEquals_UDINT(Expected:= 32, Actual:= stActual.nSize, Message:= 'Valid Slice /w length 32');

stActual := F_SpanSlice(stSpan:= stFromSpan, nStart:= 31, nLength:= 1);
AssertEquals_ULINT(Expected:= 154, Actual:= stActual.pBuffer, Message:= 'Valid Slice /w start 31');
AssertEquals_UDINT(Expected:= 1, Actual:= stActual.nSize, Message:= 'Vakud Slice /w length 1');

stActual := F_SpanSlice(stSpan:= stFromSpan, nStart:= 0, nLength:= 33);
AssertEquals_ULINT(Expected:= 123, Actual:= stActual.pBuffer, Message:= 'Invalid Slice /w start 0 - returns original');
AssertEquals_UDINT(Expected:= 32, Actual:= stActual.nSize, Message:= 'Invalid Slice /w length 33 - returns original');

stActual := F_SpanSlice(stSpan:= stFromSpan, nStart:= TO_UDINT(-1), nLength:= 32);
AssertEquals_ULINT(Expected:= 123, Actual:= stActual.pBuffer, Message:= 'Invalid Slice /w start -1 - returns original');
AssertEquals_UDINT(Expected:= 32, Actual:= stActual.nSize, Message:= 'Invalid Slice /w length 32 - returns original');

stActual := F_SpanSlice(stSpan:= stFromSpan, nStart:= 0, nLength:= TO_UDINT(-1));
AssertEquals_ULINT(Expected:= 123, Actual:= stActual.pBuffer, Message:= 'Invalid Slice /w start 0 - returns original');
AssertEquals_UDINT(Expected:= 32, Actual:= stActual.nSize, Message:= 'Invalid Slice /w length -1 - returns original');

stActual := F_SpanSlice(stSpan:= stFromSpan, nStart:= 32, nLength:= 1);
AssertEquals_ULINT(Expected:= 123, Actual:= stActual.pBuffer, Message:= 'Invalid Slice /w start 32 - returns original');
AssertEquals_UDINT(Expected:= 32, Actual:= stActual.nSize, Message:= 'Invalid Slice /w length 1 - returns original');

TEST_FINISHED_NAMED(__POUNAME());

END_FUNCTION_BLOCK

// ---- POUs/Span/F_SpanSlice.TcPOU
// Forms a slice out of the current read-only span starting at a specified index for a specified length.
FUNCTION F_SpanSlice : ST_Span
VAR_IN_OUT CONSTANT
    stSpan  : ST_SPAN;
END_VAR
VAR_INPUT
    nStart  : UDINT;        // The zero-based index at which to begin this slice.
    nLength : UDINT;        // The desired length for the slice.
END_VAR


F_SpanSlice := stSpan;

IF nStart > stSpan.nSize THEN
    RETURN;
END_IF

IF (nLength + nStart) > stSpan.nSize THEN
    RETURN;
END_IF

F_SpanSlice.pBuffer := stSpan.pBuffer + nStart;
F_SpanSlice.nSize := nLength;

END_FUNCTION

// ---- __TESTs/_ISSUES/PRG_IssuesTests.TcPOU
{attribute 'analysis' := '-33'}
PROGRAM INTERNAL PRG_IssuesTests
VAR
{IF defined (UNIT_TEST)}
	fbIssue4Tests : FB_Issue4Tests;
{END_IF}
END_VAR

END_PROGRAM

// ---- __TESTs/_ISSUES/FB_Issue4Tests.TcPOU
FUNCTION_BLOCK FINAL FB_Issue4Tests EXTENDS FB_TestSuite
VAR_INPUT
END_VAR
VAR_OUTPUT
END_VAR
VAR
	fbSutParser : FB_RepeatedEnumTests;
	fbSutWriter : FB_RepeatedEnumTests;
	stActualStruct : ST_RepeatedEnumTests;
	stExpectedStruct : ST_RepeatedEnumTests := (
		enum_values_sint_count := 5,
		enum_values_sint := [
			E_EnumOfTypeSint.VALUE_MAX,
			E_EnumOfTypeSint.VALUE_MIN,
			E_EnumOfTypeSint.VALUE_0,
			E_EnumOfTypeSint.VALUE_2,
			E_EnumOfTypeSint.VALUE_1]);
	aBuffer : ARRAY[0..63] OF BYTE;
	hrParser : HRESULT;
	hrWriter : HRESULT;
END_VAR

TEST(__POUNAME());

// Arrange
fbSutWriter.RepeatedEnumTests := stExpectedStruct;

// Act
hrWriter := fbSutWriter.Writer.WriteTo(aBuffer);
hrParser := fbSutParser.Parser.ParseFrom(aBuffer);
stActualStruct := fbSutParser.RepeatedEnumTests;

// Assert
AssertEquals_UDINT(Expected:= 8, Actual:= fbSutWriter.CalculateSize(), Message:= 'Wrong message size.');
AssertEquals_DINT(Expected:= S_OK, Actual:= hrWriter, Message:= 'Expected hrWriter = S_OK instead of error.');
AssertEquals_DINT(Expected:= S_OK, Actual:= hrParser, Message:= 'Expected hrParser = S_OK instead of error.');
AssertEquals(Expected:= stExpectedStruct, Actual:= stActualStruct, Message:= '');

TEST_FINISHED_NAMED(__POUNAME());

END_FUNCTION_BLOCK

// ---- __TESTs/_ISSUES/_gen/FB_RepeatedEnumTests.TcPOU
(*******************************************************************************
                          protoc-gen-twincat V0.0.0.0                           
                  https://github.com/TcHaxx/protoc-gen-twincat                  
*******************************************************************************)
{attribute 'no_explicit_call' := 'do not call this POU directly'}
{attribute 'no-analysis'}
FUNCTION_BLOCK INTERNAL FINAL FB_RepeatedEnumTests IMPLEMENTS I_Message
VAR
    _fbMessageParser : FB_MessageParser(ipMessage:= THIS^);
    _fbMessageWriter : FB_MessageWriter(ipMessage:= THIS^);
    _stRepeatedEnumTests : ST_RepeatedEnumTests;
    // repeated EnumOfTypeSint enum_values_sint = 1;
    _fbFieldCodecId1 : FB_FieldCodecEnum(nTag:= 16#0A);
    _fbRepeatedId1 : FB_RepeatedField(anyArray:= F_ToAnyType(_stRepeatedEnumTests.enum_values_sint), anyFirstElem:= F_ToAnyType(_stRepeatedEnumTests.enum_values_sint[0]), ipFieldCodec:= _fbFieldCodecId1);
    END_VAR

